    movel([0.119411, -1.390472, -2.566228, -0.755689, 1.570796, 1.690207],accel_mss,speed_ms,0,blend_radius_m)
    movel([0.119247, -1.390171, -2.566445, -0.755774, 1.570796, 1.690044],accel_mss,speed_ms,0,blend_radius_m)
    movel([0.119299, -1.389742, -2.566752, -0.755894, 1.570796, 1.690095],accel_mss,speed_ms,0,blend_radius_m)
    movel([0.119560, -1.389145, -2.567181, -0.756063, 1.570796, 1.690357],accel_mss,speed_ms,0,blend_radius_m)
    movel([0.120675, -1.387270, -2.568525, -0.756595, 1.570796, 1.691472],accel_mss,speed_ms,0,blend_radius_m)
    movel([0.122734, -1.387703, -2.568215, -0.756471, 1.570796, 1.693530],accel_mss,speed_ms,0,blend_radius_m)
    speed_ms = 0.005
    # Splitting Linear movement in 4 (instruction 341: MoveL 309)
    movel([0.122734, -1.385520, -2.567229, -0.759641, 1.570796, 1.693530],accel_mss,speed_ms,0,blend_radius_m)
    movel([0.122734, -1.383346, -2.566239, -0.762804, 1.570796, 1.693530],accel_mss,speed_ms,0,blend_radius_m)
    movel([0.122734, -1.381182, -2.565245, -0.765961, 1.570796, 1.693530],accel_mss,speed_ms,0,blend_radius_m)
    movel([0.122734, -1.379028, -2.564248, -0.769113, 1.570796, 1.693530],accel_mss,speed_ms,0,blend_radius_m)
    speed_ms = 0.040
    # Splitting Linear movement in 18 (instruction 343: MoveL 310)
    movel([0.125073, -1.377791, -2.565121, -0.769477, 1.570796, 1.695869],accel_mss,speed_ms,0,blend_radius_m)
    movel([0.127416, -1.376554, -2.565991, -0.769844, 1.570796, 1.698212],accel_mss,speed_ms,0,blend_radius_m)
    movel([0.129763, -1.375318, -2.566858, -0.770212, 1.570796, 1.700560],accel_mss,speed_ms,0,blend_radius_m)
    movel([0.132116, -1.374083, -2.567723, -0.770583, 1.570796, 1.702912],accel_mss,speed_ms,0,blend_radius_m)
    movel([0.134472, -1.372849, -2.568585, -0.770955, 1.570796, 1.705269],accel_mss,speed_ms,0,blend_radius_m)
    movel([0.136834, -1.371616, -2.569444, -0.771330, 1.570796, 1.707630],accel_mss,speed_ms,0,blend_radius_m)
    movel([0.139200, -1.370383, -2.570300, -0.771706, 1.570796, 1.709996],accel_mss,speed_ms,0,blend_radius_m)
    movel([0.141570, -1.369152, -2.571153, -0.772084, 1.570796, 1.712366],accel_mss,speed_ms,0,blend_radius_m)
    movel([0.143945, -1.367921, -2.572004, -0.772464, 1.570796, 1.714741],accel_mss,speed_ms,0,blend_radius_m)
    movel([0.146324, -1.366692, -2.572852, -0.772845, 1.570796, 1.717121],accel_mss,speed_ms,0,blend_radius_m)
    movel([0.148708, -1.365463, -2.573697, -0.773229, 1.570796, 1.719505],accel_mss,speed_ms,0,blend_radius_m)
    movel([0.151097, -1.364235, -2.574540, -0.773614, 1.570796, 1.721893],accel_mss,speed_ms,0,blend_radius_m)
    movel([0.153490, -1.363008, -2.575379, -0.774001, 1.570796, 1.724286],accel_mss,speed_ms,0,blend_radius_m)
    movel([0.155887, -1.361783, -2.576216, -0.774390, 1.570796, 1.726684],accel_mss,speed_ms,0,blend_radius_m)
    movel([0.158289, -1.360558, -2.577050, -0.774781, 1.570796, 1.729086],accel_mss,speed_ms,0,blend_radius_m)
    movel([0.160696, -1.359335, -2.577881, -0.775173, 1.570796, 1.731492],accel_mss,speed_ms,0,blend_radius_m)
    movel([0.163106, -1.358112, -2.578709, -0.775568, 1.570796, 1.733903],accel_mss,speed_ms,0,blend_radius_m)
    movel([0.165522, -1.356891, -2.579535, -0.775963, 1.570796, 1.736318],accel_mss,speed_ms,0,blend_radius_m)
    speed_ms = 0.005
    # Splitting Linear movement in 6 (instruction 345: MoveL 311)
    movel([0.165522, -1.358351, -2.580216, -0.773822, 1.570796, 1.736318],accel_mss,speed_ms,0,blend_radius_m)
    movel([0.165522, -1.359815, -2.580896, -0.771678, 1.570796, 1.736318],accel_mss,speed_ms,0,blend_radius_m)
    movel([0.165522, -1.361284, -2.581574, -0.769531, 1.570796, 1.736318],accel_mss,speed_ms,0,blend_radius_m)
    movel([0.165522, -1.362758, -2.582250, -0.767381, 1.570796, 1.736318],accel_mss,speed_ms,0,blend_radius_m)
    movel([0.165522, -1.364236, -2.582925, -0.765228, 1.570796, 1.736318],accel_mss,speed_ms,0,blend_radius_m)
    movel([0.165522, -1.365719, -2.583598, -0.763072, 1.570796, 1.736318],accel_mss,speed_ms,0,blend_radius_m)
    speed_ms = 0.035
    movel([0.167244, -1.365978, -2.583421, -0.762990, 1.570796, 1.738040],accel_mss,speed_ms,0,blend_radius_m)
    movel([0.168585, -1.365976, -2.583423, -0.762991, 1.570796, 1.739382],accel_mss,speed_ms,0,blend_radius_m)
    movel([0.169955, -1.365852, -2.583507, -0.763030, 1.570796, 1.740751],accel_mss,speed_ms,0,blend_radius_m)
    movel([0.171344, -1.365613, -2.583670, -0.763105, 1.570796, 1.742141],accel_mss,speed_ms,0,blend_radius_m)
    movel([0.172746, -1.365263, -2.583910, -0.763216, 1.570796, 1.743542],accel_mss,speed_ms,0,blend_radius_m)
    movel([0.174155, -1.364806, -2.584222, -0.763361, 1.570796, 1.744951],accel_mss,speed_ms,0,blend_radius_m)
    movel([0.176950, -1.363591, -2.585050, -0.763747, 1.570796, 1.747746],accel_mss,speed_ms,0,blend_radius_m)
    movel([0.178323, -1.362842, -2.585561, -0.763987, 1.570796, 1.749120],accel_mss,speed_ms,0,blend_radius_m)
    movel([0.180981, -1.361082, -2.586755, -0.764552, 1.570796, 1.751777],accel_mss,speed_ms,0,blend_radius_m)
    movel([0.182252, -1.360079, -2.587434, -0.764876, 1.570796, 1.753048],accel_mss,speed_ms,0,blend_radius_m)
    movel([0.184624, -1.357854, -2.588935, -0.765600, 1.570796, 1.755420],accel_mss,speed_ms,0,blend_radius_m)
    movel([0.185715, -1.356638, -2.589752, -0.765999, 1.570796, 1.756511],accel_mss,speed_ms,0,blend_radius_m)
    movel([0.186729, -1.355358, -2.590610, -0.766421, 1.570796, 1.757525],accel_mss,speed_ms,0,blend_radius_m)
    movel([0.187656, -1.354022, -2.591503, -0.766863, 1.570796, 1.758453],accel_mss,speed_ms,0,blend_radius_m)
    movel([0.188445, -1.352706, -2.592381, -0.767302, 1.570796, 1.759241],accel_mss,speed_ms,0,blend_radius_m)
    movel([0.189111, -1.351390, -2.593256, -0.767743, 1.570796, 1.759907],accel_mss,speed_ms,0,blend_radius_m)
    movel([0.190069, -1.348792, -2.594976, -0.768621, 1.570796, 1.760866],accel_mss,speed_ms,0,blend_radius_m)
    movel([0.190366, -1.347523, -2.595813, -0.769053, 1.570796, 1.761162],accel_mss,speed_ms,0,blend_radius_m)
    movel([0.190585, -1.345090, -2.597412, -0.769888, 1.570796, 1.761381],accel_mss,speed_ms,0,blend_radius_m)
    movel([0.190509, -1.343939, -2.598165, -0.770285, 1.570796, 1.761306],accel_mss,speed_ms,0,blend_radius_m)
    movel([0.189997, -1.341806, -2.599556, -0.771027, 1.570796, 1.760793],accel_mss,speed_ms,0,blend_radius_m)
    movel([0.189557, -1.340837, -2.600186, -0.771366, 1.570796, 1.760353],accel_mss,speed_ms,0,blend_radius_m)
    movel([0.188317, -1.339142, -2.601284, -0.771962, 1.570796, 1.759113],accel_mss,speed_ms,0,blend_radius_m)
    movel([0.187516, -1.338431, -2.601744, -0.772214, 1.570796, 1.758312],accel_mss,speed_ms,0,blend_radius_m)
    movel([0.186599, -1.337819, -2.602140, -0.772431, 1.570796, 1.757395],accel_mss,speed_ms,0,blend_radius_m)
    movel([0.185562, -1.337314, -2.602465, -0.772610, 1.570796, 1.756358],accel_mss,speed_ms,0,blend_radius_m)
    movel([0.183890, -1.336813, -2.602788, -0.772788, 1.570796, 1.754686],accel_mss,speed_ms,0,blend_radius_m)
    movel([0.183257, -1.336822, -2.602782, -0.772785, 1.570796, 1.754053],accel_mss,speed_ms,0,blend_radius_m)
    movel([0.182728, -1.337024, -2.602652, -0.772713, 1.570796, 1.753524],accel_mss,speed_ms,0,blend_radius_m)
    movel([0.182274, -1.337436, -2.602386, -0.772567, 1.570796, 1.753070],accel_mss,speed_ms,0,blend_radius_m)
    movel([0.181874, -1.338070, -2.601977, -0.772342, 1.570796, 1.752671],accel_mss,speed_ms,0,blend_radius_m)
    movel([0.181131, -1.340075, -2.600680, -0.771634, 1.570796, 1.751927],accel_mss,speed_ms,0,blend_radius_m)
    movel([0.182746, -1.340641, -2.600313, -0.771435, 1.570796, 1.753542],accel_mss,speed_ms,0,blend_radius_m)
    movel([0.184246, -1.341473, -2.599772, -0.771144, 1.570796, 1.755043],accel_mss,speed_ms,0,blend_radius_m)
    movel([0.185396, -1.342588, -2.599046, -0.770754, 1.570796, 1.756192],accel_mss,speed_ms,0,blend_radius_m)
    movel([0.186193, -1.343946, -2.598160, -0.770283, 1.570796, 1.756989],accel_mss,speed_ms,0,blend_radius_m)
    movel([0.186629, -1.345508, -2.597137, -0.769744, 1.570796, 1.757425],accel_mss,speed_ms,0,blend_radius_m)
    movel([0.186702, -1.347235, -2.596002, -0.769151, 1.570796, 1.757498],accel_mss,speed_ms,0,blend_radius_m)
    movel([0.186412, -1.349088, -2.594781, -0.768520, 1.570796, 1.757208],accel_mss,speed_ms,0,blend_radius_m)
    movel([0.185753, -1.351031, -2.593494, -0.767864, 1.570796, 1.756550],accel_mss,speed_ms,0,blend_radius_m)
    movel([0.184722, -1.353022, -2.592171, -0.767197, 1.570796, 1.755519],accel_mss,speed_ms,0,blend_radius_m)
    movel([0.183346, -1.354989, -2.590857, -0.766543, 1.570796, 1.754142],accel_mss,speed_ms,0,blend_radius_m)
    movel([0.181729, -1.356786, -2.589652, -0.765950, 1.570796, 1.752525],accel_mss,speed_ms,0,blend_radius_m)
    movel([0.179917, -1.358392, -2.588573, -0.765425, 1.570796, 1.750714],accel_mss,speed_ms,0,blend_radius_m)
    movel([0.177958, -1.359777, -2.587638, -0.764974, 1.570796, 1.748754],accel_mss,speed_ms,0,blend_radius_m)
    movel([0.175895, -1.360914, -2.586869, -0.764606, 1.570796, 1.746691],accel_mss,speed_ms,0,blend_radius_m)
    movel([0.173775, -1.361775, -2.586285, -0.764329, 1.570796, 1.744572],accel_mss,speed_ms,0,blend_radius_m)
    movel([0.171644, -1.362334, -2.585905, -0.764149, 1.570796, 1.742441],accel_mss,speed_ms,0,blend_radius_m)
    movel([0.169547, -1.362562, -2.585751, -0.764076, 1.570796, 1.740343],accel_mss,speed_ms,0,blend_radius_m)
    movel([0.167897, -1.362665, -2.585681, -0.764043, 1.570796, 1.738693],accel_mss,speed_ms,0,blend_radius_m)
    movel([0.167339, -1.362805, -2.585585, -0.763998, 1.570796, 1.738135],accel_mss,speed_ms,0,blend_radius_m)
    movel([0.166903, -1.363048, -2.585420, -0.763921, 1.570796, 1.737699],accel_mss,speed_ms,0,blend_radius_m)
    movel([0.166548, -1.363425, -2.585164, -0.763800, 1.570796, 1.737344],accel_mss,speed_ms,0,blend_radius_m)
    movel([0.166226, -1.363977, -2.584788, -0.763625, 1.570796, 1.737022],accel_mss,speed_ms,0,blend_radius_m)
    movel([0.165522, -1.365719, -2.583598, -0.763072, 1.570796, 1.736318],accel_mss,speed_ms,0,blend_radius_m)
    movel([0.167244, -1.365978, -2.583421, -0.762990, 1.570796, 1.738040],accel_mss,speed_ms,0,blend_radius_m)
    movel([0.167727, -1.365979, -2.583420, -0.762990, 1.570796, 1.738523],accel_mss,speed_ms,0,blend_radius_m)
    speed_ms = 0.005
    # Splitting Linear movement in 4 (instruction 405: MoveL 369)
    movel([0.167727, -1.363756, -2.582411, -0.766222, 1.570796, 1.738523],accel_mss,speed_ms,0,blend_radius_m)
    movel([0.167727, -1.361544, -2.581397, -0.769448, 1.570796, 1.738523],accel_mss,speed_ms,0,blend_radius_m)
    movel([0.167727, -1.359343, -2.580380, -0.772667, 1.570796, 1.738523],accel_mss,speed_ms,0,blend_radius_m)
    movel([0.167727, -1.357152, -2.579359, -0.775879, 1.570796, 1.738523],accel_mss,speed_ms,0,blend_radius_m)
    speed_ms = 0.040
    # Splitting Linear movement in 6 (instruction 407: MoveL 370)
    movel([0.165743, -1.356725, -2.579647, -0.776017, 1.570796, 1.736539],accel_mss,speed_ms,0,blend_radius_m)
    movel([0.163755, -1.356303, -2.579931, -0.776155, 1.570796, 1.734551],accel_mss,speed_ms,0,blend_radius_m)
    movel([0.161764, -1.355886, -2.580213, -0.776291, 1.570796, 1.732560],accel_mss,speed_ms,0,blend_radius_m)
    movel([0.159768, -1.355473, -2.580491, -0.776426, 1.570796, 1.730565],accel_mss,speed_ms,0,blend_radius_m)
    movel([0.157769, -1.355064, -2.580766, -0.776559, 1.570796, 1.728566],accel_mss,speed_ms,0,blend_radius_m)
    movel([0.155767, -1.354660, -2.581037, -0.776692, 1.570796, 1.726563],accel_mss,speed_ms,0,blend_radius_m)
    speed_ms = 0.005
    # Splitting Linear movement in 6 (instruction 409: MoveL 371)
    movel([0.155767, -1.356122, -2.581720, -0.774547, 1.570796, 1.726563],accel_mss,speed_ms,0,blend_radius_m)
    movel([0.155767, -1.357589, -2.582401, -0.772398, 1.570796, 1.726563],accel_mss,speed_ms,0,blend_radius_m)
    movel([0.155767, -1.359061, -2.583081, -0.770247, 1.570796, 1.726563],accel_mss,speed_ms,0,blend_radius_m)
    movel([0.155767, -1.360537, -2.583759, -0.768093, 1.570796, 1.726563],accel_mss,speed_ms,0,blend_radius_m)
    movel([0.155767, -1.362018, -2.584435, -0.765935, 1.570796, 1.726563],accel_mss,speed_ms,0,blend_radius_m)
    movel([0.155767, -1.363504, -2.585110, -0.763775, 1.570796, 1.726563],accel_mss,speed_ms,0,blend_radius_m)
    speed_ms = 0.035
    movel([0.157355, -1.360742, -2.586986, -0.764662, 1.570796, 1.728151],accel_mss,speed_ms,0,blend_radius_m)
    movel([0.158736, -1.358054, -2.588800, -0.765535, 1.570796, 1.729532],accel_mss,speed_ms,0,blend_radius_m)
    movel([0.159906, -1.355440, -2.590555, -0.766394, 1.570796, 1.730702],accel_mss,speed_ms,0,blend_radius_m)
    movel([0.160863, -1.352902, -2.592250, -0.767237, 1.570796, 1.731660],accel_mss,speed_ms,0,blend_radius_m)
    movel([0.161608, -1.350441, -2.593885, -0.768063, 1.570796, 1.732405],accel_mss,speed_ms,0,blend_radius_m)
    movel([0.162137, -1.348053, -2.595464, -0.768872, 1.570796, 1.732933],accel_mss,speed_ms,0,blend_radius_m)
    movel([0.162447, -1.345744, -2.596983, -0.769663, 1.570796, 1.733244],accel_mss,speed_ms,0,blend_radius_m)
    movel([0.162537, -1.343514, -2.598442, -0.770433, 1.570796, 1.733334],accel_mss,speed_ms,0,blend_radius_m)
    movel([0.162403, -1.341361, -2.599845, -0.771183, 1.570796, 1.733200],accel_mss,speed_ms,0,blend_radius_m)
    movel([0.162046, -1.339287, -2.601191, -0.771911, 1.570796, 1.732842],accel_mss,speed_ms,0,blend_radius_m)
    movel([0.161461, -1.337295, -2.602477, -0.772617, 1.570796, 1.732257],accel_mss,speed_ms,0,blend_radius_m)
    movel([0.160647, -1.335385, -2.603706, -0.773298, 1.570796, 1.731443],accel_mss,speed_ms,0,blend_radius_m)
    movel([0.159603, -1.333559, -2.604876, -0.773954, 1.570796, 1.730399],accel_mss,speed_ms,0,blend_radius_m)
    movel([0.158326, -1.331816, -2.605989, -0.774584, 1.570796, 1.729123],accel_mss,speed_ms,0,blend_radius_m)
    movel([0.156817, -1.330161, -2.607041, -0.775187, 1.570796, 1.727613],accel_mss,speed_ms,0,blend_radius_m)
    movel([0.155070, -1.328593, -2.608035, -0.775761, 1.570796, 1.725866],accel_mss,speed_ms,0,blend_radius_m)
    movel([0.156422, -1.327583, -2.608673, -0.776133, 1.570796, 1.727219],accel_mss,speed_ms,0,blend_radius_m)
    movel([0.158344, -1.325960, -2.609696, -0.776733, 1.570796, 1.729140],accel_mss,speed_ms,0,blend_radius_m)
    movel([0.160279, -1.327317, -2.608841, -0.776231, 1.570796, 1.731076],accel_mss,speed_ms,0,blend_radius_m)
    movel([0.161946, -1.328931, -2.607821, -0.775637, 1.570796, 1.732742],accel_mss,speed_ms,0,blend_radius_m)
    movel([0.163339, -1.330774, -2.606652, -0.774963, 1.570796, 1.734136],accel_mss,speed_ms,0,blend_radius_m)
    movel([0.164467, -1.332824, -2.605345, -0.774219, 1.570796, 1.735263],accel_mss,speed_ms,0,blend_radius_m)
    movel([0.165329, -1.335051, -2.603920, -0.773418, 1.570796, 1.736126],accel_mss,speed_ms,0,blend_radius_m)
    movel([0.165930, -1.337434, -2.602388, -0.772567, 1.570796, 1.736726],accel_mss,speed_ms,0,blend_radius_m)
    movel([0.166274, -1.339941, -2.600767, -0.771681, 1.570796, 1.737070],accel_mss,speed_ms,0,blend_radius_m)
    movel([0.166364, -1.342551, -2.599071, -0.770767, 1.570796, 1.737160],accel_mss,speed_ms,0,blend_radius_m)
    movel([0.166202, -1.345238, -2.597314, -0.769836, 1.570796, 1.736998],accel_mss,speed_ms,0,blend_radius_m)
    movel([0.165795, -1.347977, -2.595514, -0.768898, 1.570796, 1.736591],accel_mss,speed_ms,0,blend_radius_m)
    movel([0.165144, -1.350747, -2.593682, -0.767959, 1.570796, 1.735940],accel_mss,speed_ms,0,blend_radius_m)
    movel([0.164254, -1.353520, -2.591838, -0.767031, 1.570796, 1.735050],accel_mss,speed_ms,0,blend_radius_m)
    movel([0.163128, -1.356279, -2.589993, -0.766117, 1.570796, 1.733924],accel_mss,speed_ms,0,blend_radius_m)
    movel([0.161769, -1.358997, -2.588164, -0.765227, 1.570796, 1.732566],accel_mss,speed_ms,0,blend_radius_m)
    movel([0.160179, -1.361655, -2.586367, -0.764368, 1.570796, 1.730976],accel_mss,speed_ms,0,blend_radius_m)
    movel([0.158366, -1.364231, -2.584614, -0.763544, 1.570796, 1.729162],accel_mss,speed_ms,0,blend_radius_m)
    movel([0.155767, -1.363504, -2.585110, -0.763775, 1.570796, 1.726563],accel_mss,speed_ms,0,blend_radius_m)
    movel([0.157104, -1.361176, -2.586691, -0.764522, 1.570796, 1.727901],accel_mss,speed_ms,0,blend_radius_m)
    speed_ms = 0.005
    # Splitting Linear movement in 6 (instruction 448: MoveL 408)
    movel([0.157104, -1.359687, -2.586015, -0.766687, 1.570796, 1.727901],accel_mss,speed_ms,0,blend_radius_m)
    movel([0.157104, -1.358204, -2.585337, -0.768848, 1.570796, 1.727901],accel_mss,speed_ms,0,blend_radius_m)
    movel([0.157104, -1.356725, -2.584657, -0.771007, 1.570796, 1.727901],accel_mss,speed_ms,0,blend_radius_m)
    movel([0.157104, -1.355250, -2.583976, -0.773162, 1.570796, 1.727901],accel_mss,speed_ms,0,blend_radius_m)
    movel([0.157104, -1.353781, -2.583293, -0.775315, 1.570796, 1.727901],accel_mss,speed_ms,0,blend_radius_m)
    movel([0.157104, -1.352316, -2.582608, -0.777465, 1.570796, 1.727901],accel_mss,speed_ms,0,blend_radius_m)
    speed_ms = 0.040
    # Splitting Linear movement in 6 (instruction 450: MoveL 409)
    movel([0.154683, -1.352853, -2.582249, -0.777287, 1.570796, 1.725480],accel_mss,speed_ms,0,blend_radius_m)
    movel([0.152263, -1.353395, -2.581886, -0.777108, 1.570796, 1.723059],accel_mss,speed_ms,0,blend_radius_m)
    movel([0.149843, -1.353940, -2.581520, -0.776928, 1.570796, 1.720639],accel_mss,speed_ms,0,blend_radius_m)
    movel([0.147424, -1.354490, -2.581151, -0.776747, 1.570796, 1.718220],accel_mss,speed_ms,0,blend_radius_m)
    movel([0.145005, -1.355044, -2.580779, -0.776566, 1.570796, 1.715801],accel_mss,speed_ms,0,blend_radius_m)
    movel([0.142587, -1.355603, -2.580403, -0.776383, 1.570796, 1.713383],accel_mss,speed_ms,0,blend_radius_m)
    speed_ms = 0.005
    # Splitting Linear movement in 6 (instruction 452: MoveL 410)
    movel([0.142587, -1.357064, -2.581085, -0.774240, 1.570796, 1.713383],accel_mss,speed_ms,0,blend_radius_m)
    movel([0.142587, -1.358530, -2.581766, -0.772093, 1.570796, 1.713383],accel_mss,speed_ms,0,blend_radius_m)
    movel([0.142587, -1.360001, -2.582445, -0.769944, 1.570796, 1.713383],accel_mss,speed_ms,0,blend_radius_m)
    movel([0.142587, -1.361476, -2.583122, -0.767791, 1.570796, 1.713383],accel_mss,speed_ms,0,blend_radius_m)
    movel([0.142587, -1.362956, -2.583798, -0.765636, 1.570796, 1.713383],accel_mss,speed_ms,0,blend_radius_m)
    movel([0.142587, -1.364440, -2.584472, -0.763477, 1.570796, 1.713383],accel_mss,speed_ms,0,blend_radius_m)
    speed_ms = 0.035
    movel([0.144618, -1.363400, -2.585181, -0.763808, 1.570796, 1.715414],accel_mss,speed_ms,0,blend_radius_m)
    movel([0.145265, -1.363158, -2.585346, -0.763886, 1.570796, 1.716061],accel_mss,speed_ms,0,blend_radius_m)
    movel([0.145714, -1.363112, -2.585377, -0.763900, 1.570796, 1.716510],accel_mss,speed_ms,0,blend_radius_m)
    movel([0.146013, -1.363264, -2.585273, -0.763852, 1.570796, 1.716810],accel_mss,speed_ms,0,blend_radius_m)
    movel([0.146199, -1.363626, -2.585027, -0.763736, 1.570796, 1.716996],accel_mss,speed_ms,0,blend_radius_m)
    movel([0.146391, -1.364992, -2.584095, -0.763302, 1.570796, 1.717188],accel_mss,speed_ms,0,blend_radius_m)
    movel([0.146678, -1.366931, -2.582768, -0.762690, 1.570796, 1.717475],accel_mss,speed_ms,0,blend_radius_m)
    movel([0.147186, -1.368743, -2.581523, -0.762123, 1.570796, 1.717982],accel_mss,speed_ms,0,blend_radius_m)
    movel([0.147904, -1.370420, -2.580367, -0.761602, 1.570796, 1.718700],accel_mss,speed_ms,0,blend_radius_m)
    movel([0.148823, -1.371955, -2.579305, -0.761129, 1.570796, 1.719620],accel_mss,speed_ms,0,blend_radius_m)
    movel([0.149928, -1.373343, -2.578342, -0.760705, 1.570796, 1.720724],accel_mss,speed_ms,0,blend_radius_m)
    movel([0.151213, -1.374577, -2.577483, -0.760329, 1.570796, 1.722009],accel_mss,speed_ms,0,blend_radius_m)
    movel([0.152668, -1.375652, -2.576733, -0.760004, 1.570796, 1.723464],accel_mss,speed_ms,0,blend_radius_m)
    movel([0.154279, -1.376563, -2.576096, -0.759729, 1.570796, 1.725075],accel_mss,speed_ms,0,blend_radius_m)
    movel([0.156039, -1.377302, -2.575579, -0.759508, 1.570796, 1.726835],accel_mss,speed_ms,0,blend_radius_m)
    movel([0.157942, -1.377860, -2.575188, -0.759341, 1.570796, 1.728738],accel_mss,speed_ms,0,blend_radius_m)
    movel([0.159972, -1.378236, -2.574924, -0.759229, 1.570796, 1.730769],accel_mss,speed_ms,0,blend_radius_m)
    movel([0.162127, -1.378415, -2.574799, -0.759176, 1.570796, 1.732924],accel_mss,speed_ms,0,blend_radius_m)
    movel([0.164395, -1.378396, -2.574812, -0.759181, 1.570796, 1.735192],accel_mss,speed_ms,0,blend_radius_m)
    movel([0.166771, -1.378169, -2.574971, -0.759249, 1.570796, 1.737567],accel_mss,speed_ms,0,blend_radius_m)
    movel([0.169243, -1.377725, -2.575282, -0.759381, 1.570796, 1.740039],accel_mss,speed_ms,0,blend_radius_m)
    movel([0.171807, -1.377058, -2.575750, -0.759581, 1.570796, 1.742603],accel_mss,speed_ms,0,blend_radius_m)
    movel([0.174557, -1.376132, -2.576398, -0.759859, 1.570796, 1.745353],accel_mss,speed_ms,0,blend_radius_m)
    movel([0.177244, -1.375031, -2.577167, -0.760192, 1.570796, 1.748040],accel_mss,speed_ms,0,blend_radius_m)
    movel([0.179860, -1.373766, -2.578047, -0.760576, 1.570796, 1.750657],accel_mss,speed_ms,0,blend_radius_m)
    movel([0.182392, -1.372346, -2.579033, -0.761009, 1.570796, 1.753189],accel_mss,speed_ms,0,blend_radius_m)
    movel([0.184834, -1.370780, -2.580118, -0.761491, 1.570796, 1.755630],accel_mss,speed_ms,0,blend_radius_m)
    movel([0.187171, -1.369080, -2.581291, -0.762018, 1.570796, 1.757967],accel_mss,speed_ms,0,blend_radius_m)
    movel([0.189395, -1.367255, -2.582546, -0.762588, 1.570796, 1.760191],accel_mss,speed_ms,0,blend_radius_m)
    movel([0.191497, -1.365311, -2.583877, -0.763201, 1.570796, 1.762293],accel_mss,speed_ms,0,blend_radius_m)
    movel([0.193462, -1.363263, -2.585274, -0.763852, 1.570796, 1.764258],accel_mss,speed_ms,0,blend_radius_m)
    movel([0.195284, -1.361118, -2.586730, -0.764540, 1.570796, 1.766080],accel_mss,speed_ms,0,blend_radius_m)
    movel([0.196947, -1.358890, -2.588237, -0.765262, 1.570796, 1.767743],accel_mss,speed_ms,0,blend_radius_m)
    movel([0.198441, -1.356584, -2.589788, -0.766017, 1.570796, 1.769238],accel_mss,speed_ms,0,blend_radius_m)
    movel([0.199751, -1.354218, -2.591373, -0.766799, 1.570796, 1.770547],accel_mss,speed_ms,0,blend_radius_m)
    movel([0.200870, -1.351797, -2.592986, -0.767607, 1.570796, 1.771666],accel_mss,speed_ms,0,blend_radius_m)
    movel([0.201780, -1.349333, -2.594619, -0.768437, 1.570796, 1.772576],accel_mss,speed_ms,0,blend_radius_m)
    movel([0.202469, -1.346842, -2.596261, -0.769286, 1.570796, 1.773266],accel_mss,speed_ms,0,blend_radius_m)
    movel([0.202849, -1.344806, -2.597598, -0.769986, 1.570796, 1.773645],accel_mss,speed_ms,0,blend_radius_m)
    movel([0.203044, -1.342836, -2.598885, -0.770668, 1.570796, 1.773841],accel_mss,speed_ms,0,blend_radius_m)
    movel([0.203058, -1.340938, -2.600120, -0.771331, 1.570796, 1.773854],accel_mss,speed_ms,0,blend_radius_m)
    movel([0.202894, -1.339124, -2.601296, -0.771969, 1.570796, 1.773690],accel_mss,speed_ms,0,blend_radius_m)
    movel([0.202553, -1.337396, -2.602412, -0.772581, 1.570796, 1.773349],accel_mss,speed_ms,0,blend_radius_m)
    movel([0.202041, -1.335767, -2.603461, -0.773161, 1.570796, 1.772837],accel_mss,speed_ms,0,blend_radius_m)
    movel([0.201360, -1.334242, -2.604439, -0.773708, 1.570796, 1.772156],accel_mss,speed_ms,0,blend_radius_m)
    movel([0.200513, -1.332830, -2.605342, -0.774217, 1.570796, 1.771309],accel_mss,speed_ms,0,blend_radius_m)
    movel([0.199505, -1.331537, -2.606166, -0.774686, 1.570796, 1.770301],accel_mss,speed_ms,0,blend_radius_m)
    movel([0.198339, -1.330373, -2.606906, -0.775110, 1.570796, 1.769136],accel_mss,speed_ms,0,blend_radius_m)
    movel([0.197021, -1.329344, -2.607559, -0.775486, 1.570796, 1.767817],accel_mss,speed_ms,0,blend_radius_m)
    movel([0.195555, -1.328459, -2.608119, -0.775810, 1.570796, 1.766352],accel_mss,speed_ms,0,blend_radius_m)
    movel([0.193946, -1.327726, -2.608583, -0.776080, 1.570796, 1.764742],accel_mss,speed_ms,0,blend_radius_m)
    movel([0.192197, -1.327150, -2.608947, -0.776293, 1.570796, 1.762993],accel_mss,speed_ms,0,blend_radius_m)
    movel([0.190314, -1.326740, -2.609205, -0.776444, 1.570796, 1.761110],accel_mss,speed_ms,0,blend_radius_m)
    movel([0.188302, -1.326505, -2.609353, -0.776531, 1.570796, 1.759098],accel_mss,speed_ms,0,blend_radius_m)
    movel([0.186033, -1.326287, -2.609490, -0.776612, 1.570796, 1.756829],accel_mss,speed_ms,0,blend_radius_m)
    movel([0.186699, -1.324329, -2.610721, -0.777339, 1.570796, 1.757495],accel_mss,speed_ms,0,blend_radius_m)
    movel([0.187062, -1.323682, -2.611126, -0.777581, 1.570796, 1.757858],accel_mss,speed_ms,0,blend_radius_m)
    movel([0.187486, -1.323227, -2.611411, -0.777751, 1.570796, 1.758283],accel_mss,speed_ms,0,blend_radius_m)
    movel([0.188004, -1.322935, -2.611594, -0.777861, 1.570796, 1.758800],accel_mss,speed_ms,0,blend_radius_m)
    movel([0.188643, -1.322782, -2.611689, -0.777918, 1.570796, 1.759439],accel_mss,speed_ms,0,blend_radius_m)
    movel([0.190414, -1.322802, -2.611676, -0.777910, 1.570796, 1.761210],accel_mss,speed_ms,0,blend_radius_m)
    movel([0.192754, -1.323116, -2.611480, -0.777793, 1.570796, 1.763550],accel_mss,speed_ms,0,blend_radius_m)
    movel([0.194935, -1.323635, -2.611155, -0.777598, 1.570796, 1.765732],accel_mss,speed_ms,0,blend_radius_m)
    movel([0.196955, -1.324350, -2.610707, -0.777331, 1.570796, 1.767752],accel_mss,speed_ms,0,blend_radius_m)
    movel([0.198804, -1.325254, -2.610140, -0.776995, 1.570796, 1.769600],accel_mss,speed_ms,0,blend_radius_m)
    movel([0.200476, -1.326336, -2.609459, -0.776593, 1.570796, 1.771272],accel_mss,speed_ms,0,blend_radius_m)
    movel([0.201971, -1.327585, -2.608672, -0.776132, 1.570796, 1.772767],accel_mss,speed_ms,0,blend_radius_m)
    movel([0.203277, -1.328995, -2.607780, -0.775614, 1.570796, 1.774073],accel_mss,speed_ms,0,blend_radius_m)
    movel([0.204395, -1.330550, -2.606794, -0.775045, 1.570796, 1.775192],accel_mss,speed_ms,0,blend_radius_m)
    movel([0.205318, -1.332246, -2.605714, -0.774428, 1.570796, 1.776115],accel_mss,speed_ms,0,blend_radius_m)
    movel([0.206044, -1.334068, -2.604550, -0.773771, 1.570796, 1.776841],accel_mss,speed_ms,0,blend_radius_m)
    movel([0.206568, -1.336009, -2.603305, -0.773075, 1.570796, 1.777365],accel_mss,speed_ms,0,blend_radius_m)
    movel([0.206883, -1.338059, -2.601984, -0.772345, 1.570796, 1.777680],accel_mss,speed_ms,0,blend_radius_m)
    movel([0.206991, -1.340206, -2.600596, -0.771588, 1.570796, 1.777788],accel_mss,speed_ms,0,blend_radius_m)
    movel([0.206884, -1.342444, -2.599140, -0.770805, 1.570796, 1.777681],accel_mss,speed_ms,0,blend_radius_m)
    movel([0.206563, -1.344758, -2.597629, -0.770002, 1.570796, 1.777359],accel_mss,speed_ms,0,blend_radius_m)
    movel([0.206022, -1.347143, -2.596063, -0.769183, 1.570796, 1.776818],accel_mss,speed_ms,0,blend_radius_m)
    movel([0.205270, -1.349550, -2.594475, -0.768364, 1.570796, 1.776066],accel_mss,speed_ms,0,blend_radius_m)
    movel([0.204329, -1.351941, -2.592890, -0.767558, 1.570796, 1.775125],accel_mss,speed_ms,0,blend_radius_m)
    movel([0.203206, -1.354307, -2.591313, -0.766769, 1.570796, 1.774003],accel_mss,speed_ms,0,blend_radius_m)
    movel([0.201915, -1.356634, -2.589755, -0.766000, 1.570796, 1.772711],accel_mss,speed_ms,0,blend_radius_m)
    movel([0.200464, -1.358916, -2.588219, -0.765254, 1.570796, 1.771260],accel_mss,speed_ms,0,blend_radius_m)
    movel([0.198867, -1.361141, -2.586715, -0.764533, 1.570796, 1.769664],accel_mss,speed_ms,0,blend_radius_m)
    movel([0.197131, -1.363302, -2.585247, -0.763839, 1.570796, 1.767927],accel_mss,speed_ms,0,blend_radius_m)
    movel([0.195269, -1.365387, -2.583825, -0.763177, 1.570796, 1.766065],accel_mss,speed_ms,0,blend_radius_m)
    movel([0.193289, -1.367390, -2.582453, -0.762546, 1.570796, 1.764085],accel_mss,speed_ms,0,blend_radius_m)
    movel([0.191199, -1.369302, -2.581138, -0.761949, 1.570796, 1.761995],accel_mss,speed_ms,0,blend_radius_m)
    movel([0.189008, -1.371111, -2.579889, -0.761389, 1.570796, 1.759805],accel_mss,speed_ms,0,blend_radius_m)
    movel([0.186730, -1.372813, -2.578709, -0.760866, 1.570796, 1.757527],accel_mss,speed_ms,0,blend_radius_m)
    movel([0.184369, -1.374394, -2.577610, -0.760385, 1.570796, 1.755166],accel_mss,speed_ms,0,blend_radius_m)
    movel([0.181935, -1.375853, -2.576593, -0.759943, 1.570796, 1.752731],accel_mss,speed_ms,0,blend_radius_m)
    movel([0.179436, -1.377174, -2.575669, -0.759546, 1.570796, 1.750233],accel_mss,speed_ms,0,blend_radius_m)
    movel([0.176882, -1.378351, -2.574844, -0.759195, 1.570796, 1.747678],accel_mss,speed_ms,0,blend_radius_m)
    movel([0.174330, -1.379357, -2.574136, -0.758895, 1.570796, 1.745127],accel_mss,speed_ms,0,blend_radius_m)
    movel([0.171808, -1.380183, -2.573555, -0.758651, 1.570796, 1.742604],accel_mss,speed_ms,0,blend_radius_m)
    movel([0.169325, -1.380833, -2.573097, -0.758460, 1.570796, 1.740121],accel_mss,speed_ms,0,blend_radius_m)
    movel([0.166894, -1.381304, -2.572764, -0.758321, 1.570796, 1.737691],accel_mss,speed_ms,0,blend_radius_m)
    movel([0.164518, -1.381602, -2.572553, -0.758233, 1.570796, 1.735315],accel_mss,speed_ms,0,blend_radius_m)
    movel([0.162212, -1.381729, -2.572463, -0.758196, 1.570796, 1.733009],accel_mss,speed_ms,0,blend_radius_m)
    movel([0.159981, -1.381688, -2.572493, -0.758208, 1.570796, 1.730778],accel_mss,speed_ms,0,blend_radius_m)
    movel([0.157837, -1.381474, -2.572644, -0.758271, 1.570796, 1.728633],accel_mss,speed_ms,0,blend_radius_m)
    movel([0.155786, -1.381095, -2.572911, -0.758382, 1.570796, 1.726582],accel_mss,speed_ms,0,blend_radius_m)
    movel([0.153843, -1.380549, -2.573297, -0.758543, 1.570796, 1.724639],accel_mss,speed_ms,0,blend_radius_m)
    movel([0.152016, -1.379836, -2.573800, -0.758754, 1.570796, 1.722813],accel_mss,speed_ms,0,blend_radius_m)
    movel([0.150314, -1.378957, -2.574418, -0.759014, 1.570796, 1.721111],accel_mss,speed_ms,0,blend_radius_m)
    movel([0.148748, -1.377914, -2.575150, -0.759325, 1.570796, 1.719545],accel_mss,speed_ms,0,blend_radius_m)
    movel([0.147329, -1.376704, -2.575998, -0.759687, 1.570796, 1.718125],accel_mss,speed_ms,0,blend_radius_m)
    movel([0.146068, -1.375329, -2.576959, -0.760101, 1.570796, 1.716865],accel_mss,speed_ms,0,blend_radius_m)
    movel([0.144973, -1.373788, -2.578032, -0.760569, 1.570796, 1.715770],accel_mss,speed_ms,0,blend_radius_m)
    movel([0.143879, -1.371725, -2.579464, -0.761200, 1.570796, 1.714675],accel_mss,speed_ms,0,blend_radius_m)
    movel([0.143082, -1.369495, -2.581005, -0.761889, 1.570796, 1.713878],accel_mss,speed_ms,0,blend_radius_m)
    movel([0.142634, -1.367074, -2.582670, -0.762645, 1.570796, 1.713430],accel_mss,speed_ms,0,blend_radius_m)
    movel([0.142587, -1.364440, -2.584472, -0.763477, 1.570796, 1.713383],accel_mss,speed_ms,0,blend_radius_m)
    movel([0.144618, -1.363400, -2.585181, -0.763808, 1.570796, 1.715414],accel_mss,speed_ms,0,blend_radius_m)
    movel([0.145130, -1.363209, -2.585311, -0.763869, 1.570796, 1.715926],accel_mss,speed_ms,0,blend_radius_m)
    speed_ms = 0.005
    # Splitting Linear movement in 4 (instruction 570: MoveL 526)
    movel([0.145130, -1.360982, -2.584298, -0.767110, 1.570796, 1.715926],accel_mss,speed_ms,0,blend_radius_m)
    movel([0.145130, -1.358765, -2.583281, -0.770343, 1.570796, 1.715926],accel_mss,speed_ms,0,blend_radius_m)
    movel([0.145130, -1.356559, -2.582261, -0.773569, 1.570796, 1.715926],accel_mss,speed_ms,0,blend_radius_m)
    movel([0.145130, -1.354363, -2.581237, -0.776789, 1.570796, 1.715926],accel_mss,speed_ms,0,blend_radius_m)
    speed_ms = 0.040
    # Splitting Linear movement in 10 (instruction 572: MoveL 527)
    movel([0.142834, -1.354927, -2.580858, -0.776604, 1.570796, 1.713630],accel_mss,speed_ms,0,blend_radius_m)
    movel([0.140539, -1.355494, -2.580476, -0.776419, 1.570796, 1.711335],accel_mss,speed_ms,0,blend_radius_m)
    movel([0.138244, -1.356065, -2.580092, -0.776232, 1.570796, 1.709040],accel_mss,speed_ms,0,blend_radius_m)
    movel([0.135951, -1.356640, -2.579704, -0.776045, 1.570796, 1.706747],accel_mss,speed_ms,0,blend_radius_m)
    movel([0.133658, -1.357218, -2.579314, -0.775857, 1.570796, 1.704454],accel_mss,speed_ms,0,blend_radius_m)
    movel([0.131366, -1.357800, -2.578921, -0.775669, 1.570796, 1.702162],accel_mss,speed_ms,0,blend_radius_m)
    movel([0.129075, -1.358385, -2.578525, -0.775479, 1.570796, 1.699871],accel_mss,speed_ms,0,blend_radius_m)
    movel([0.126784, -1.358974, -2.578126, -0.775289, 1.570796, 1.697581],accel_mss,speed_ms,0,blend_radius_m)
    movel([0.124495, -1.359567, -2.577724, -0.775099, 1.570796, 1.695291],accel_mss,speed_ms,0,blend_radius_m)
    movel([0.122207, -1.360163, -2.577319, -0.774908, 1.570796, 1.693003],accel_mss,speed_ms,0,blend_radius_m)
    speed_ms = 0.005
    # Splitting Linear movement in 4 (instruction 574: MoveL 528)
    movel([0.122207, -1.362349, -2.578336, -0.771704, 1.570796, 1.693003],accel_mss,speed_ms,0,blend_radius_m)
    movel([0.122207, -1.364545, -2.579350, -0.768493, 1.570796, 1.693003],accel_mss,speed_ms,0,blend_radius_m)
    movel([0.122207, -1.366752, -2.580361, -0.765276, 1.570796, 1.693003],accel_mss,speed_ms,0,blend_radius_m)
    movel([0.122207, -1.368969, -2.581367, -0.762053, 1.570796, 1.693003],accel_mss,speed_ms,0,blend_radius_m)
    speed_ms = 0.035
    movel([0.120628, -1.371920, -2.579329, -0.761140, 1.570796, 1.691424],accel_mss,speed_ms,0,blend_radius_m)
    movel([0.119214, -1.371762, -2.579438, -0.761188, 1.570796, 1.690010],accel_mss,speed_ms,0,blend_radius_m)
    movel([0.117940, -1.371473, -2.579638, -0.761277, 1.570796, 1.688737],accel_mss,speed_ms,0,blend_radius_m)
    movel([0.116802, -1.371057, -2.579926, -0.761406, 1.570796, 1.687599],accel_mss,speed_ms,0,blend_radius_m)
    movel([0.115794, -1.370517, -2.580299, -0.761572, 1.570796, 1.686590],accel_mss,speed_ms,0,blend_radius_m)
    movel([0.114907, -1.369857, -2.580755, -0.761777, 1.570796, 1.685704],accel_mss,speed_ms,0,blend_radius_m)
    movel([0.114139, -1.369082, -2.581290, -0.762018, 1.570796, 1.684935],accel_mss,speed_ms,0,blend_radius_m)
    movel([0.113482, -1.368197, -2.581899, -0.762294, 1.570796, 1.684278],accel_mss,speed_ms,0,blend_radius_m)
    movel([0.112927, -1.367203, -2.582581, -0.762605, 1.570796, 1.683724],accel_mss,speed_ms,0,blend_radius_m)
    movel([0.112291, -1.365333, -2.583862, -0.763194, 1.570796, 1.683087],accel_mss,speed_ms,0,blend_radius_m)
    movel([0.112068, -1.363283, -2.585260, -0.763846, 1.570796, 1.682864],accel_mss,speed_ms,0,blend_radius_m)
    movel([0.112247, -1.361095, -2.586746, -0.764548, 1.570796, 1.683043],accel_mss,speed_ms,0,blend_radius_m)
    movel([0.112813, -1.358816, -2.588287, -0.765286, 1.570796, 1.683610],accel_mss,speed_ms,0,blend_radius_m)
    movel([0.113756, -1.356481, -2.589857, -0.766050, 1.570796, 1.684553],accel_mss,speed_ms,0,blend_radius_m)
    movel([0.115059, -1.354143, -2.591423, -0.766823, 1.570796, 1.685855],accel_mss,speed_ms,0,blend_radius_m)
    movel([0.116712, -1.351839, -2.592957, -0.767592, 1.570796, 1.687508],accel_mss,speed_ms,0,blend_radius_m)
    movel([0.118694, -1.349622, -2.594428, -0.768340, 1.570796, 1.689491],accel_mss,speed_ms,0,blend_radius_m)
    movel([0.120927, -1.347589, -2.595769, -0.769030, 1.570796, 1.691723],accel_mss,speed_ms,0,blend_radius_m)
    movel([0.123311, -1.345817, -2.596935, -0.769637, 1.570796, 1.694107],accel_mss,speed_ms,0,blend_radius_m)
    movel([0.125806, -1.344321, -2.597915, -0.770153, 1.570796, 1.696602],accel_mss,speed_ms,0,blend_radius_m)
    movel([0.128360, -1.343128, -2.598694, -0.770567, 1.570796, 1.699157],accel_mss,speed_ms,0,blend_radius_m)
    movel([0.130924, -1.342257, -2.599262, -0.770870, 1.570796, 1.701720],accel_mss,speed_ms,0,blend_radius_m)
    movel([0.133454, -1.341729, -2.599606, -0.771054, 1.570796, 1.704250],accel_mss,speed_ms,0,blend_radius_m)
    movel([0.135896, -1.341564, -2.599713, -0.771112, 1.570796, 1.706692],accel_mss,speed_ms,0,blend_radius_m)
    movel([0.138205, -1.341781, -2.599572, -0.771036, 1.570796, 1.709002],accel_mss,speed_ms,0,blend_radius_m)
    movel([0.140282, -1.342388, -2.599177, -0.770824, 1.570796, 1.711078],accel_mss,speed_ms,0,blend_radius_m)
    movel([0.142032, -1.343350, -2.598549, -0.770489, 1.570796, 1.712829],accel_mss,speed_ms,0,blend_radius_m)
    movel([0.143439, -1.344635, -2.597709, -0.770045, 1.570796, 1.714235],accel_mss,speed_ms,0,blend_radius_m)
    movel([0.144488, -1.346208, -2.596678, -0.769503, 1.570796, 1.715284],accel_mss,speed_ms,0,blend_radius_m)
    movel([0.145165, -1.348036, -2.595475, -0.768878, 1.570796, 1.715961],accel_mss,speed_ms,0,blend_radius_m)
    movel([0.145455, -1.350083, -2.594123, -0.768184, 1.570796, 1.716251],accel_mss,speed_ms,0,blend_radius_m)
    movel([0.145344, -1.352316, -2.592640, -0.767432, 1.570796, 1.716141],accel_mss,speed_ms,0,blend_radius_m)
    movel([0.144824, -1.354700, -2.591050, -0.766639, 1.570796, 1.715620],accel_mss,speed_ms,0,blend_radius_m)
    movel([0.144168, -1.356513, -2.589836, -0.766040, 1.570796, 1.714964],accel_mss,speed_ms,0,blend_radius_m)
    movel([0.143799, -1.357128, -2.589423, -0.765838, 1.570796, 1.714595],accel_mss,speed_ms,0,blend_radius_m)
    movel([0.143353, -1.357588, -2.589114, -0.765687, 1.570796, 1.714149],accel_mss,speed_ms,0,blend_radius_m)
    movel([0.142793, -1.357923, -2.588888, -0.765578, 1.570796, 1.713589],accel_mss,speed_ms,0,blend_radius_m)
    movel([0.142084, -1.358161, -2.588728, -0.765500, 1.570796, 1.712880],accel_mss,speed_ms,0,blend_radius_m)
    movel([0.140076, -1.358461, -2.588526, -0.765402, 1.570796, 1.710872],accel_mss,speed_ms,0,blend_radius_m)
    movel([0.140788, -1.355200, -2.590716, -0.766473, 1.570796, 1.711585],accel_mss,speed_ms,0,blend_radius_m)
    movel([0.141097, -1.352421, -2.592571, -0.767398, 1.570796, 1.711893],accel_mss,speed_ms,0,blend_radius_m)
    movel([0.140994, -1.350112, -2.594103, -0.768174, 1.570796, 1.711790],accel_mss,speed_ms,0,blend_radius_m)
    movel([0.140462, -1.348263, -2.595325, -0.768801, 1.570796, 1.711258],accel_mss,speed_ms,0,blend_radius_m)
    movel([0.140033, -1.347506, -2.595824, -0.769059, 1.570796, 1.710829],accel_mss,speed_ms,0,blend_radius_m)
    movel([0.139494, -1.346858, -2.596251, -0.769280, 1.570796, 1.710290],accel_mss,speed_ms,0,blend_radius_m)
    movel([0.138842, -1.346318, -2.596606, -0.769465, 1.570796, 1.709638],accel_mss,speed_ms,0,blend_radius_m)
    movel([0.137202, -1.345554, -2.597107, -0.769728, 1.570796, 1.707998],accel_mss,speed_ms,0,blend_radius_m)
    movel([0.136209, -1.345326, -2.597257, -0.769806, 1.570796, 1.707005],accel_mss,speed_ms,0,blend_radius_m)
    movel([0.133874, -1.345167, -2.597361, -0.769861, 1.570796, 1.704670],accel_mss,speed_ms,0,blend_radius_m)
    movel([0.131737, -1.345382, -2.597220, -0.769787, 1.570796, 1.702534],accel_mss,speed_ms,0,blend_radius_m)
    movel([0.129547, -1.345948, -2.596849, -0.769593, 1.570796, 1.700343],accel_mss,speed_ms,0,blend_radius_m)
    movel([0.127354, -1.346830, -2.596269, -0.769290, 1.570796, 1.698150],accel_mss,speed_ms,0,blend_radius_m)
    movel([0.125210, -1.347998, -2.595500, -0.768891, 1.570796, 1.696007],accel_mss,speed_ms,0,blend_radius_m)
    movel([0.123173, -1.349416, -2.594564, -0.768409, 1.570796, 1.693969],accel_mss,speed_ms,0,blend_radius_m)
    movel([0.121287, -1.351053, -2.593479, -0.767856, 1.570796, 1.692083],accel_mss,speed_ms,0,blend_radius_m)
    movel([0.119605, -1.352873, -2.592270, -0.767246, 1.570796, 1.690401],accel_mss,speed_ms,0,blend_radius_m)
    movel([0.118176, -1.354846, -2.590953, -0.766590, 1.570796, 1.688972],accel_mss,speed_ms,0,blend_radius_m)
    movel([0.116876, -1.357206, -2.589370, -0.765812, 1.570796, 1.687673],accel_mss,speed_ms,0,blend_radius_m)
    movel([0.116086, -1.359360, -2.587920, -0.765109, 1.570796, 1.686883],accel_mss,speed_ms,0,blend_radius_m)
    movel([0.115884, -1.360363, -2.587241, -0.764784, 1.570796, 1.686680],accel_mss,speed_ms,0,blend_radius_m)
    movel([0.115866, -1.362242, -2.585968, -0.764179, 1.570796, 1.686662],accel_mss,speed_ms,0,blend_radius_m)
    movel([0.116049, -1.363120, -2.585371, -0.763898, 1.570796, 1.686846],accel_mss,speed_ms,0,blend_radius_m)
    movel([0.116806, -1.364762, -2.584252, -0.763375, 1.570796, 1.687602],accel_mss,speed_ms,0,blend_radius_m)
    movel([0.118084, -1.366274, -2.583218, -0.762897, 1.570796, 1.688880],accel_mss,speed_ms,0,blend_radius_m)
    movel([0.119883, -1.367669, -2.582262, -0.762459, 1.570796, 1.690680],accel_mss,speed_ms,0,blend_radius_m)
    movel([0.122207, -1.368969, -2.581367, -0.762053, 1.570796, 1.693003],accel_mss,speed_ms,0,blend_radius_m)
    movel([0.120970, -1.371277, -2.579774, -0.761338, 1.570796, 1.691767],accel_mss,speed_ms,0,blend_radius_m)
    speed_ms = 0.005
    # Splitting Linear movement in 6 (instruction 644: MoveL 596)
    movel([0.120970, -1.369801, -2.579105, -0.763483, 1.570796, 1.691767],accel_mss,speed_ms,0,blend_radius_m)
    movel([0.120970, -1.368329, -2.578435, -0.765626, 1.570796, 1.691767],accel_mss,speed_ms,0,blend_radius_m)
    movel([0.120970, -1.366861, -2.577762, -0.767765, 1.570796, 1.691767],accel_mss,speed_ms,0,blend_radius_m)
    movel([0.120970, -1.365398, -2.577088, -0.769902, 1.570796, 1.691767],accel_mss,speed_ms,0,blend_radius_m)
    movel([0.120970, -1.363940, -2.576413, -0.772036, 1.570796, 1.691767],accel_mss,speed_ms,0,blend_radius_m)
    movel([0.120970, -1.362487, -2.575736, -0.774167, 1.570796, 1.691767],accel_mss,speed_ms,0,blend_radius_m)
    speed_ms = 0.040
    # Splitting Linear movement in 18 (instruction 646: MoveL 597)
    movel([0.120281, -1.360880, -2.576831, -0.774678, 1.570796, 1.691078],accel_mss,speed_ms,0,blend_radius_m)
    movel([0.119589, -1.359271, -2.577924, -0.775194, 1.570796, 1.690386],accel_mss,speed_ms,0,blend_radius_m)
    movel([0.118894, -1.357660, -2.579015, -0.775714, 1.570796, 1.689691],accel_mss,speed_ms,0,blend_radius_m)
    movel([0.118196, -1.356047, -2.580104, -0.776238, 1.570796, 1.688993],accel_mss,speed_ms,0,blend_radius_m)
    movel([0.117496, -1.354432, -2.581190, -0.776767, 1.570796, 1.688292],accel_mss,speed_ms,0,blend_radius_m)
    movel([0.116792, -1.352815, -2.582275, -0.777299, 1.570796, 1.687588],accel_mss,speed_ms,0,blend_radius_m)
    movel([0.116085, -1.351195, -2.583357, -0.777837, 1.570796, 1.686882],accel_mss,speed_ms,0,blend_radius_m)
    movel([0.115376, -1.349574, -2.584437, -0.778378, 1.570796, 1.686172],accel_mss,speed_ms,0,blend_radius_m)
    movel([0.114663, -1.347950, -2.585515, -0.778924, 1.570796, 1.685460],accel_mss,speed_ms,0,blend_radius_m)
    movel([0.113948, -1.346324, -2.586591, -0.779475, 1.570796, 1.684744],accel_mss,speed_ms,0,blend_radius_m)
    movel([0.113229, -1.344696, -2.587664, -0.780029, 1.570796, 1.684025],accel_mss,speed_ms,0,blend_radius_m)
    movel([0.112508, -1.343065, -2.588736, -0.780588, 1.570796, 1.683304],accel_mss,speed_ms,0,blend_radius_m)
    movel([0.111783, -1.341433, -2.589805, -0.781152, 1.570796, 1.682579],accel_mss,speed_ms,0,blend_radius_m)
    movel([0.111055, -1.339798, -2.590871, -0.781719, 1.570796, 1.681852],accel_mss,speed_ms,0,blend_radius_m)
    movel([0.110324, -1.338161, -2.591936, -0.782292, 1.570796, 1.681121],accel_mss,speed_ms,0,blend_radius_m)
    movel([0.109590, -1.336522, -2.592998, -0.782868, 1.570796, 1.680387],accel_mss,speed_ms,0,blend_radius_m)
    movel([0.108853, -1.334881, -2.594059, -0.783449, 1.570796, 1.679650],accel_mss,speed_ms,0,blend_radius_m)
    movel([0.108113, -1.333238, -2.595116, -0.784034, 1.570796, 1.678910],accel_mss,speed_ms,0,blend_radius_m)
    speed_ms = 0.005
    # Splitting Linear movement in 6 (instruction 648: MoveL 598)
    movel([0.108113, -1.334723, -2.595815, -0.781850, 1.570796, 1.678910],accel_mss,speed_ms,0,blend_radius_m)
    movel([0.108113, -1.336214, -2.596512, -0.779663, 1.570796, 1.678910],accel_mss,speed_ms,0,blend_radius_m)
    movel([0.108113, -1.337709, -2.597208, -0.777473, 1.570796, 1.678910],accel_mss,speed_ms,0,blend_radius_m)
    movel([0.108113, -1.339209, -2.597901, -0.775279, 1.570796, 1.678910],accel_mss,speed_ms,0,blend_radius_m)
    movel([0.108113, -1.340714, -2.598593, -0.773082, 1.570796, 1.678910],accel_mss,speed_ms,0,blend_radius_m)
    movel([0.108113, -1.342224, -2.599284, -0.770881, 1.570796, 1.678910],accel_mss,speed_ms,0,blend_radius_m)
    speed_ms = 0.035
    movel([0.106316, -1.344176, -2.598009, -0.770203, 1.570796, 1.677112],accel_mss,speed_ms,0,blend_radius_m)
    movel([0.104661, -1.346139, -2.596723, -0.769527, 1.570796, 1.675458],accel_mss,speed_ms,0,blend_radius_m)
    movel([0.103151, -1.348105, -2.595429, -0.768854, 1.570796, 1.673947],accel_mss,speed_ms,0,blend_radius_m)
    movel([0.101779, -1.350073, -2.594129, -0.768187, 1.570796, 1.672575],accel_mss,speed_ms,0,blend_radius_m)
    movel([0.100547, -1.352034, -2.592828, -0.767527, 1.570796, 1.671344],accel_mss,speed_ms,0,blend_radius_m)
    movel([0.099454, -1.353987, -2.591527, -0.766875, 1.570796, 1.670250],accel_mss,speed_ms,0,blend_radius_m)
    movel([0.098494, -1.355925, -2.590231, -0.766234, 1.570796, 1.669290],accel_mss,speed_ms,0,blend_radius_m)
    movel([0.097668, -1.357843, -2.588942, -0.765604, 1.570796, 1.668464],accel_mss,speed_ms,0,blend_radius_m)
    movel([0.096975, -1.359738, -2.587665, -0.764987, 1.570796, 1.667771],accel_mss,speed_ms,0,blend_radius_m)
    movel([0.096414, -1.361603, -2.586402, -0.764384, 1.570796, 1.667210],accel_mss,speed_ms,0,blend_radius_m)
    movel([0.095669, -1.365229, -2.583933, -0.763227, 1.570796, 1.666466],accel_mss,speed_ms,0,blend_radius_m)
    movel([0.095485, -1.366984, -2.582732, -0.762673, 1.570796, 1.666281],accel_mss,speed_ms,0,blend_radius_m)
    movel([0.095485, -1.370347, -2.580417, -0.761625, 1.570796, 1.666281],accel_mss,speed_ms,0,blend_radius_m)
    movel([0.095663, -1.371951, -2.579308, -0.761131, 1.570796, 1.666459],accel_mss,speed_ms,0,blend_radius_m)
    movel([0.096371, -1.374980, -2.577202, -0.760207, 1.570796, 1.667167],accel_mss,speed_ms,0,blend_radius_m)
    movel([0.096895, -1.376399, -2.576211, -0.759779, 1.570796, 1.667692],accel_mss,speed_ms,0,blend_radius_m)
    movel([0.098286, -1.379018, -2.574375, -0.758996, 1.570796, 1.669082],accel_mss,speed_ms,0,blend_radius_m)
    movel([0.099145, -1.380214, -2.573533, -0.758642, 1.570796, 1.669941],accel_mss,speed_ms,0,blend_radius_m)
    movel([0.101187, -1.382355, -2.572020, -0.758013, 1.570796, 1.671984],accel_mss,speed_ms,0,blend_radius_m)
    movel([0.102370, -1.383294, -2.571355, -0.757739, 1.570796, 1.673166],accel_mss,speed_ms,0,blend_radius_m)
    movel([0.103656, -1.384139, -2.570755, -0.757494, 1.570796, 1.674453],accel_mss,speed_ms,0,blend_radius_m)
    movel([0.105046, -1.384888, -2.570223, -0.757278, 1.570796, 1.675842],accel_mss,speed_ms,0,blend_radius_m)
    movel([0.106539, -1.385533, -2.569764, -0.757092, 1.570796, 1.677335],accel_mss,speed_ms,0,blend_radius_m)
    movel([0.108133, -1.386075, -2.569377, -0.756936, 1.570796, 1.678929],accel_mss,speed_ms,0,blend_radius_m)
    movel([0.109829, -1.386506, -2.569070, -0.756813, 1.570796, 1.680626],accel_mss,speed_ms,0,blend_radius_m)
    movel([0.111627, -1.386823, -2.568843, -0.756722, 1.570796, 1.682423],accel_mss,speed_ms,0,blend_radius_m)
    movel([0.113523, -1.387023, -2.568701, -0.756665, 1.570796, 1.684320],accel_mss,speed_ms,0,blend_radius_m)
    movel([0.112735, -1.388822, -2.567413, -0.756154, 1.570796, 1.683531],accel_mss,speed_ms,0,blend_radius_m)
    movel([0.112369, -1.389479, -2.566941, -0.755968, 1.570796, 1.683166],accel_mss,speed_ms,0,blend_radius_m)
    movel([0.111916, -1.389894, -2.566643, -0.755852, 1.570796, 1.682713],accel_mss,speed_ms,0,blend_radius_m)
    movel([0.111348, -1.390097, -2.566497, -0.755795, 1.570796, 1.682144],accel_mss,speed_ms,0,blend_radius_m)
    movel([0.110638, -1.390114, -2.566485, -0.755790, 1.570796, 1.681434],accel_mss,speed_ms,0,blend_radius_m)
    movel([0.107947, -1.389760, -2.566740, -0.755889, 1.570796, 1.678743],accel_mss,speed_ms,0,blend_radius_m)
    movel([0.105434, -1.389150, -2.567177, -0.756061, 1.570796, 1.676230],accel_mss,speed_ms,0,blend_radius_m)
    movel([0.103104, -1.388299, -2.567788, -0.756302, 1.570796, 1.673901],accel_mss,speed_ms,0,blend_radius_m)
    movel([0.100967, -1.387215, -2.568564, -0.756610, 1.570796, 1.671763],accel_mss,speed_ms,0,blend_radius_m)
    movel([0.099025, -1.385916, -2.569491, -0.756982, 1.570796, 1.669822],accel_mss,speed_ms,0,blend_radius_m)
    movel([0.097291, -1.384409, -2.570564, -0.757416, 1.570796, 1.668087],accel_mss,speed_ms,0,blend_radius_m)
    movel([0.095771, -1.382708, -2.571771, -0.757910, 1.570796, 1.666568],accel_mss,speed_ms,0,blend_radius_m)
    movel([0.094473, -1.380827, -2.573100, -0.758461, 1.570796, 1.665270],accel_mss,speed_ms,0,blend_radius_m)
    movel([0.093411, -1.378773, -2.574547, -0.759069, 1.570796, 1.664208],accel_mss,speed_ms,0,blend_radius_m)
    movel([0.092590, -1.376560, -2.576099, -0.759730, 1.570796, 1.663386],accel_mss,speed_ms,0,blend_radius_m)
    movel([0.092021, -1.374198, -2.577747, -0.760444, 1.570796, 1.662818],accel_mss,speed_ms,0,blend_radius_m)
    movel([0.091719, -1.371698, -2.579483, -0.761208, 1.570796, 1.662515],accel_mss,speed_ms,0,blend_radius_m)
    movel([0.091688, -1.369075, -2.581294, -0.762020, 1.570796, 1.662485],accel_mss,speed_ms,0,blend_radius_m)
    movel([0.091943, -1.366340, -2.583173, -0.762876, 1.570796, 1.662739],accel_mss,speed_ms,0,blend_radius_m)
    movel([0.092496, -1.363503, -2.585110, -0.763775, 1.570796, 1.663292],accel_mss,speed_ms,0,blend_radius_m)
    movel([0.093354, -1.360578, -2.587096, -0.764715, 1.570796, 1.664150],accel_mss,speed_ms,0,blend_radius_m)
    movel([0.095047, -1.356318, -2.589967, -0.766104, 1.570796, 1.665843],accel_mss,speed_ms,0,blend_radius_m)
    movel([0.096067, -1.354205, -2.591381, -0.766803, 1.570796, 1.666864],accel_mss,speed_ms,0,blend_radius_m)
    movel([0.097206, -1.352103, -2.592782, -0.767504, 1.570796, 1.668002],accel_mss,speed_ms,0,blend_radius_m)
    movel([0.098471, -1.350011, -2.594170, -0.768208, 1.570796, 1.669267],accel_mss,speed_ms,0,blend_radius_m)
    movel([0.099865, -1.347930, -2.595545, -0.768914, 1.570796, 1.670662],accel_mss,speed_ms,0,blend_radius_m)
    movel([0.101395, -1.345856, -2.596909, -0.769624, 1.570796, 1.672192],accel_mss,speed_ms,0,blend_radius_m)
    movel([0.103062, -1.343793, -2.598260, -0.770336, 1.570796, 1.673858],accel_mss,speed_ms,0,blend_radius_m)
    movel([0.104534, -1.342128, -2.599346, -0.770915, 1.570796, 1.675330],accel_mss,speed_ms,0,blend_radius_m)
    movel([0.105082, -1.341653, -2.599655, -0.771081, 1.570796, 1.675878],accel_mss,speed_ms,0,blend_radius_m)
    movel([0.105579, -1.341395, -2.599823, -0.771171, 1.570796, 1.676375],accel_mss,speed_ms,0,blend_radius_m)
    movel([0.106077, -1.341339, -2.599860, -0.771190, 1.570796, 1.676873],accel_mss,speed_ms,0,blend_radius_m)
    movel([0.106628, -1.341469, -2.599775, -0.771145, 1.570796, 1.677424],accel_mss,speed_ms,0,blend_radius_m)
    movel([0.108113, -1.342224, -2.599284, -0.770881, 1.570796, 1.678910],accel_mss,speed_ms,0,blend_radius_m)
    movel([0.106316, -1.344176, -2.598009, -0.770203, 1.570796, 1.677112],accel_mss,speed_ms,0,blend_radius_m)
    movel([0.106109, -1.344420, -2.597850, -0.770119, 1.570796, 1.676906],accel_mss,speed_ms,0,blend_radius_m)
    speed_ms = 0.005
    # Splitting Linear movement in 6 (instruction 714: MoveL 662)
    movel([0.106109, -1.342913, -2.597161, -0.772315, 1.570796, 1.676906],accel_mss,speed_ms,0,blend_radius_m)
    movel([0.106109, -1.341410, -2.596471, -0.774508, 1.570796, 1.676906],accel_mss,speed_ms,0,blend_radius_m)
    movel([0.106109, -1.339913, -2.595778, -0.776698, 1.570796, 1.676906],accel_mss,speed_ms,0,blend_radius_m)
    movel([0.106109, -1.338420, -2.595085, -0.778884, 1.570796, 1.676906],accel_mss,speed_ms,0,blend_radius_m)
    movel([0.106109, -1.336932, -2.594389, -0.781068, 1.570796, 1.676906],accel_mss,speed_ms,0,blend_radius_m)
    movel([0.106109, -1.335449, -2.593692, -0.783248, 1.570796, 1.676906],accel_mss,speed_ms,0,blend_radius_m)
    speed_ms = 0.040
    # Splitting Linear movement in 20 (instruction 716: MoveL 663)
    movel([0.106875, -1.333194, -2.595145, -0.784050, 1.570796, 1.677671],accel_mss,speed_ms,0,blend_radius_m)
    movel([0.107644, -1.330931, -2.596596, -0.784862, 1.570796, 1.678441],accel_mss,speed_ms,0,blend_radius_m)
    movel([0.108418, -1.328659, -2.598045, -0.785685, 1.570796, 1.679214],accel_mss,speed_ms,0,blend_radius_m)
    movel([0.109195, -1.326380, -2.599493, -0.786517, 1.570796, 1.679991],accel_mss,speed_ms,0,blend_radius_m)
    movel([0.109976, -1.324091, -2.600939, -0.787359, 1.570796, 1.680773],accel_mss,speed_ms,0,blend_radius_m)
    movel([0.110761, -1.321795, -2.602383, -0.788211, 1.570796, 1.681558],accel_mss,speed_ms,0,blend_radius_m)
    movel([0.111551, -1.319489, -2.603826, -0.789074, 1.570796, 1.682347],accel_mss,speed_ms,0,blend_radius_m)
    movel([0.112344, -1.317175, -2.605267, -0.789947, 1.570796, 1.683140],accel_mss,speed_ms,0,blend_radius_m)
    movel([0.113141, -1.314853, -2.606706, -0.790830, 1.570796, 1.683938],accel_mss,speed_ms,0,blend_radius_m)
    movel([0.113943, -1.312521, -2.608144, -0.791724, 1.570796, 1.684739],accel_mss,speed_ms,0,blend_radius_m)
    movel([0.114748, -1.310181, -2.609580, -0.792628, 1.570796, 1.685545],accel_mss,speed_ms,0,blend_radius_m)
    movel([0.115558, -1.307831, -2.611014, -0.793543, 1.570796, 1.686354],accel_mss,speed_ms,0,blend_radius_m)
    movel([0.116372, -1.305473, -2.612447, -0.794469, 1.570796, 1.687168],accel_mss,speed_ms,0,blend_radius_m)
    movel([0.117190, -1.303106, -2.613878, -0.795405, 1.570796, 1.687987],accel_mss,speed_ms,0,blend_radius_m)
    movel([0.118013, -1.300729, -2.615307, -0.796353, 1.570796, 1.688809],accel_mss,speed_ms,0,blend_radius_m)
    movel([0.118839, -1.298344, -2.616734, -0.797311, 1.570796, 1.689636],accel_mss,speed_ms,0,blend_radius_m)
    movel([0.119671, -1.295949, -2.618160, -0.798281, 1.570796, 1.690467],accel_mss,speed_ms,0,blend_radius_m)
    movel([0.120506, -1.293544, -2.619583, -0.799261, 1.570796, 1.691302],accel_mss,speed_ms,0,blend_radius_m)
    movel([0.121346, -1.291130, -2.621005, -0.800253, 1.570796, 1.692142],accel_mss,speed_ms,0,blend_radius_m)
    movel([0.122190, -1.288707, -2.622426, -0.801257, 1.570796, 1.692987],accel_mss,speed_ms,0,blend_radius_m)
    speed_ms = 0.005
    # Splitting Linear movement in 4 (instruction 718: MoveL 664)
    movel([0.122190, -1.291002, -2.623523, -0.797864, 1.570796, 1.692987],accel_mss,speed_ms,0,blend_radius_m)
    movel([0.122190, -1.293310, -2.624616, -0.794463, 1.570796, 1.692987],accel_mss,speed_ms,0,blend_radius_m)
    movel([0.122190, -1.295630, -2.625706, -0.791053, 1.570796, 1.692987],accel_mss,speed_ms,0,blend_radius_m)
    movel([0.122190, -1.297963, -2.626792, -0.787634, 1.570796, 1.692987],accel_mss,speed_ms,0,blend_radius_m)
    speed_ms = 0.035
    movel([0.121345, -1.299932, -2.625623, -0.786833, 1.570796, 1.692142],accel_mss,speed_ms,0,blend_radius_m)
    movel([0.120728, -1.301794, -2.624514, -0.786081, 1.570796, 1.691524],accel_mss,speed_ms,0,blend_radius_m)
    movel([0.120340, -1.303548, -2.623464, -0.785377, 1.570796, 1.691137],accel_mss,speed_ms,0,blend_radius_m)
    movel([0.120177, -1.305199, -2.622473, -0.784718, 1.570796, 1.690973],accel_mss,speed_ms,0,blend_radius_m)
    movel([0.120238, -1.306748, -2.621539, -0.784102, 1.570796, 1.691034],accel_mss,speed_ms,0,blend_radius_m)
    movel([0.120525, -1.308197, -2.620663, -0.783529, 1.570796, 1.691322],accel_mss,speed_ms,0,blend_radius_m)
    movel([0.121039, -1.309548, -2.619843, -0.782998, 1.570796, 1.691835],accel_mss,speed_ms,0,blend_radius_m)
    movel([0.121775, -1.310804, -2.619079, -0.782506, 1.570796, 1.692571],accel_mss,speed_ms,0,blend_radius_m)
    movel([0.123160, -1.312314, -2.618158, -0.781917, 1.570796, 1.693956],accel_mss,speed_ms,0,blend_radius_m)
    movel([0.124887, -1.313419, -2.617482, -0.781488, 1.570796, 1.695683],accel_mss,speed_ms,0,blend_radius_m)
    movel([0.126906, -1.314127, -2.617048, -0.781214, 1.570796, 1.697702],accel_mss,speed_ms,0,blend_radius_m)
    movel([0.129165, -1.314438, -2.616857, -0.781093, 1.570796, 1.699961],accel_mss,speed_ms,0,blend_radius_m)
    movel([0.131624, -1.314352, -2.616910, -0.781127, 1.570796, 1.702420],accel_mss,speed_ms,0,blend_radius_m)
    movel([0.134231, -1.313872, -2.617205, -0.781313, 1.570796, 1.705027],accel_mss,speed_ms,0,blend_radius_m)
    movel([0.136947, -1.312993, -2.617743, -0.781653, 1.570796, 1.707743],accel_mss,speed_ms,0,blend_radius_m)
    movel([0.139721, -1.311711, -2.618526, -0.782151, 1.570796, 1.710517],accel_mss,speed_ms,0,blend_radius_m)
    movel([0.142427, -1.310077, -2.619521, -0.782790, 1.570796, 1.713223],accel_mss,speed_ms,0,blend_radius_m)
    movel([0.144947, -1.308172, -2.620678, -0.783539, 1.570796, 1.715744],accel_mss,speed_ms,0,blend_radius_m)
    movel([0.147248, -1.306040, -2.621966, -0.784383, 1.570796, 1.718044],accel_mss,speed_ms,0,blend_radius_m)
    movel([0.149284, -1.303726, -2.623357, -0.785306, 1.570796, 1.720081],accel_mss,speed_ms,0,blend_radius_m)
    movel([0.151023, -1.301280, -2.624821, -0.786288, 1.570796, 1.721819],accel_mss,speed_ms,0,blend_radius_m)
    movel([0.152413, -1.298752, -2.626324, -0.787312, 1.570796, 1.723209],accel_mss,speed_ms,0,blend_radius_m)
    movel([0.153421, -1.296189, -2.627841, -0.788359, 1.570796, 1.724218],accel_mss,speed_ms,0,blend_radius_m)
    movel([0.153997, -1.293642, -2.629339, -0.789407, 1.570796, 1.724793],accel_mss,speed_ms,0,blend_radius_m)
    movel([0.154134, -1.291082, -2.630837, -0.790469, 1.570796, 1.724930],accel_mss,speed_ms,0,blend_radius_m)
    movel([0.153815, -1.288798, -2.632167, -0.791424, 1.570796, 1.724612],accel_mss,speed_ms,0,blend_radius_m)
    movel([0.153057, -1.286822, -2.633311, -0.792255, 1.570796, 1.723854],accel_mss,speed_ms,0,blend_radius_m)
    movel([0.151885, -1.285181, -2.634258, -0.792949, 1.570796, 1.722682],accel_mss,speed_ms,0,blend_radius_m)
    movel([0.150315, -1.283903, -2.634993, -0.793492, 1.570796, 1.721111],accel_mss,speed_ms,0,blend_radius_m)
    movel([0.148371, -1.283016, -2.635502, -0.793870, 1.570796, 1.719168],accel_mss,speed_ms,0,blend_radius_m)
    movel([0.146077, -1.282549, -2.635770, -0.794070, 1.570796, 1.716873],accel_mss,speed_ms,0,blend_radius_m)
    movel([0.143454, -1.282525, -2.635784, -0.794080, 1.570796, 1.714250],accel_mss,speed_ms,0,blend_radius_m)
    movel([0.141686, -1.282809, -2.635621, -0.793959, 1.570796, 1.712483],accel_mss,speed_ms,0,blend_radius_m)
    movel([0.141035, -1.283059, -2.635478, -0.793852, 1.570796, 1.711832],accel_mss,speed_ms,0,blend_radius_m)
    movel([0.140530, -1.283391, -2.635287, -0.793711, 1.570796, 1.711326],accel_mss,speed_ms,0,blend_radius_m)
    movel([0.140166, -1.283807, -2.635048, -0.793533, 1.570796, 1.710962],accel_mss,speed_ms,0,blend_radius_m)
    movel([0.139936, -1.284321, -2.634753, -0.793315, 1.570796, 1.710733],accel_mss,speed_ms,0,blend_radius_m)
    movel([0.139857, -1.285655, -2.633985, -0.792749, 1.570796, 1.710654],accel_mss,speed_ms,0,blend_radius_m)
    movel([0.140062, -1.286014, -2.633778, -0.792597, 1.570796, 1.710859],accel_mss,speed_ms,0,blend_radius_m)
    movel([0.140512, -1.286275, -2.633628, -0.792487, 1.570796, 1.711308],accel_mss,speed_ms,0,blend_radius_m)
    movel([0.141094, -1.286419, -2.633545, -0.792426, 1.570796, 1.711890],accel_mss,speed_ms,0,blend_radius_m)
    movel([0.143913, -1.286469, -2.633515, -0.792404, 1.570796, 1.714709],accel_mss,speed_ms,0,blend_radius_m)
    movel([0.145854, -1.286942, -2.633242, -0.792205, 1.570796, 1.716650],accel_mss,speed_ms,0,blend_radius_m)
    movel([0.147474, -1.287813, -2.632738, -0.791838, 1.570796, 1.718271],accel_mss,speed_ms,0,blend_radius_m)
    movel([0.148747, -1.289036, -2.632029, -0.791324, 1.570796, 1.719543],accel_mss,speed_ms,0,blend_radius_m)
    movel([0.149631, -1.290566, -2.631138, -0.790684, 1.570796, 1.720427],accel_mss,speed_ms,0,blend_radius_m)
    movel([0.150095, -1.292360, -2.630091, -0.789938, 1.570796, 1.720892],accel_mss,speed_ms,0,blend_radius_m)
    movel([0.150108, -1.294370, -2.628912, -0.789107, 1.570796, 1.720905],accel_mss,speed_ms,0,blend_radius_m)
    movel([0.149938, -1.295443, -2.628281, -0.788665, 1.570796, 1.720734],accel_mss,speed_ms,0,blend_radius_m)
    movel([0.149201, -1.297760, -2.626912, -0.787716, 1.570796, 1.719997],accel_mss,speed_ms,0,blend_radius_m)
    movel([0.148659, -1.298949, -2.626208, -0.787232, 1.570796, 1.719455],accel_mss,speed_ms,0,blend_radius_m)
    movel([0.147296, -1.301249, -2.624839, -0.786301, 1.570796, 1.718093],accel_mss,speed_ms,0,blend_radius_m)
    movel([0.145613, -1.303404, -2.623550, -0.785435, 1.570796, 1.716410],accel_mss,speed_ms,0,blend_radius_m)
    movel([0.143668, -1.305367, -2.622371, -0.784651, 1.570796, 1.714464],accel_mss,speed_ms,0,blend_radius_m)
    movel([0.141512, -1.307092, -2.621331, -0.783966, 1.570796, 1.712308],accel_mss,speed_ms,0,blend_radius_m)
    movel([0.139201, -1.308533, -2.620459, -0.783397, 1.570796, 1.709997],accel_mss,speed_ms,0,blend_radius_m)
    movel([0.136788, -1.309640, -2.619788, -0.782962, 1.570796, 1.707584],accel_mss,speed_ms,0,blend_radius_m)
    movel([0.135561, -1.310054, -2.619536, -0.782799, 1.570796, 1.706357],accel_mss,speed_ms,0,blend_radius_m)
    movel([0.134326, -1.310370, -2.619344, -0.782676, 1.570796, 1.705123],accel_mss,speed_ms,0,blend_radius_m)
    movel([0.131994, -1.310660, -2.619167, -0.782562, 1.570796, 1.702791],accel_mss,speed_ms,0,blend_radius_m)
    movel([0.129883, -1.310520, -2.619252, -0.782617, 1.570796, 1.700680],accel_mss,speed_ms,0,blend_radius_m)
    movel([0.128042, -1.309974, -2.619584, -0.782831, 1.570796, 1.698839],accel_mss,speed_ms,0,blend_radius_m)
    movel([0.126514, -1.309054, -2.620143, -0.783192, 1.570796, 1.697310],accel_mss,speed_ms,0,blend_radius_m)
    movel([0.125344, -1.307792, -2.620908, -0.783689, 1.570796, 1.696140],accel_mss,speed_ms,0,blend_radius_m)
    movel([0.124583, -1.306207, -2.621865, -0.784317, 1.570796, 1.695379],accel_mss,speed_ms,0,blend_radius_m)
    movel([0.124369, -1.305304, -2.622409, -0.784676, 1.570796, 1.695165],accel_mss,speed_ms,0,blend_radius_m)
    movel([0.124274, -1.304334, -2.622992, -0.785063, 1.570796, 1.695070],accel_mss,speed_ms,0,blend_radius_m)
    movel([0.124471, -1.302193, -2.624275, -0.785921, 1.570796, 1.695267],accel_mss,speed_ms,0,blend_radius_m)
    movel([0.124610, -1.300631, -2.625207, -0.786550, 1.570796, 1.695406],accel_mss,speed_ms,0,blend_radius_m)
    movel([0.124287, -1.299454, -2.625908, -0.787027, 1.570796, 1.695083],accel_mss,speed_ms,0,blend_radius_m)
    movel([0.123483, -1.298589, -2.626421, -0.787379, 1.570796, 1.694280],accel_mss,speed_ms,0,blend_radius_m)
    movel([0.122190, -1.297963, -2.626792, -0.787634, 1.570796, 1.692987],accel_mss,speed_ms,0,blend_radius_m)
    movel([0.121345, -1.299932, -2.625623, -0.786833, 1.570796, 1.692142],accel_mss,speed_ms,0,blend_radius_m)
    movel([0.121138, -1.300559, -2.625250, -0.786580, 1.570796, 1.691935],accel_mss,speed_ms,0,blend_radius_m)
    speed_ms = 0.005
    # Splitting Linear movement in 4 (instruction 795: MoveL 739)
    movel([0.121138, -1.298230, -2.624167, -0.789992, 1.570796, 1.691935],accel_mss,speed_ms,0,blend_radius_m)
    movel([0.121138, -1.295914, -2.623080, -0.793395, 1.570796, 1.691935],accel_mss,speed_ms,0,blend_radius_m)
    movel([0.121138, -1.293609, -2.621989, -0.796790, 1.570796, 1.691935],accel_mss,speed_ms,0,blend_radius_m)
    movel([0.121138, -1.291318, -2.620895, -0.800176, 1.570796, 1.691935],accel_mss,speed_ms,0,blend_radius_m)
    speed_ms = 0.040
    # Splitting Linear movement in 10 (instruction 797: MoveL 740)
    movel([0.120168, -1.289572, -2.621919, -0.800898, 1.570796, 1.690965],accel_mss,speed_ms,0,blend_radius_m)
    movel([0.119193, -1.287825, -2.622940, -0.801624, 1.570796, 1.689990],accel_mss,speed_ms,0,blend_radius_m)
    movel([0.118214, -1.286077, -2.623958, -0.802354, 1.570796, 1.689011],accel_mss,speed_ms,0,blend_radius_m)
    movel([0.117231, -1.284326, -2.624974, -0.803089, 1.570796, 1.688027],accel_mss,speed_ms,0,blend_radius_m)
    movel([0.116242, -1.282574, -2.625986, -0.803829, 1.570796, 1.687039],accel_mss,speed_ms,0,blend_radius_m)
    movel([0.115250, -1.280820, -2.626995, -0.804573, 1.570796, 1.686046],accel_mss,speed_ms,0,blend_radius_m)
    movel([0.114252, -1.279065, -2.628002, -0.805322, 1.570796, 1.685049],accel_mss,speed_ms,0,blend_radius_m)
    movel([0.113250, -1.277308, -2.629006, -0.806076, 1.570796, 1.684047],accel_mss,speed_ms,0,blend_radius_m)
    movel([0.112244, -1.275549, -2.630006, -0.806833, 1.570796, 1.683040],accel_mss,speed_ms,0,blend_radius_m)
    movel([0.111232, -1.273789, -2.631004, -0.807596, 1.570796, 1.682029],accel_mss,speed_ms,0,blend_radius_m)
    speed_ms = 0.005
    # Splitting Linear movement in 6 (instruction 799: MoveL 741)
    movel([0.111232, -1.275331, -2.631747, -0.805311, 1.570796, 1.682029],accel_mss,speed_ms,0,blend_radius_m)
    movel([0.111232, -1.276879, -2.632489, -0.803021, 1.570796, 1.682029],accel_mss,speed_ms,0,blend_radius_m)
    movel([0.111232, -1.278433, -2.633228, -0.800728, 1.570796, 1.682029],accel_mss,speed_ms,0,blend_radius_m)
    movel([0.111232, -1.279992, -2.633967, -0.798430, 1.570796, 1.682029],accel_mss,speed_ms,0,blend_radius_m)
    movel([0.111232, -1.281557, -2.634703, -0.796129, 1.570796, 1.682029],accel_mss,speed_ms,0,blend_radius_m)
    movel([0.111232, -1.283128, -2.635438, -0.793823, 1.570796, 1.682029],accel_mss,speed_ms,0,blend_radius_m)
    speed_ms = 0.035
    movel([0.108593, -1.286019, -2.633775, -0.792595, 1.570796, 1.679389],accel_mss,speed_ms,0,blend_radius_m)
    movel([0.106209, -1.289014, -2.632042, -0.791334, 1.570796, 1.677005],accel_mss,speed_ms,0,blend_radius_m)
    movel([0.104085, -1.292083, -2.630253, -0.790053, 1.570796, 1.674882],accel_mss,speed_ms,0,blend_radius_m)
    movel([0.102227, -1.295203, -2.628422, -0.788764, 1.570796, 1.673023],accel_mss,speed_ms,0,blend_radius_m)
    movel([0.100631, -1.298351, -2.626563, -0.787476, 1.570796, 1.671427],accel_mss,speed_ms,0,blend_radius_m)
    movel([0.099307, -1.301496, -2.624692, -0.786201, 1.570796, 1.670103],accel_mss,speed_ms,0,blend_radius_m)
    movel([0.098254, -1.304622, -2.622819, -0.784948, 1.570796, 1.669050],accel_mss,speed_ms,0,blend_radius_m)
    movel([0.097473, -1.307701, -2.620963, -0.783725, 1.570796, 1.668269],accel_mss,speed_ms,0,blend_radius_m)
    movel([0.096969, -1.310714, -2.619134, -0.782541, 1.570796, 1.667765],accel_mss,speed_ms,0,blend_radius_m)
    movel([0.096738, -1.313642, -2.617346, -0.781402, 1.570796, 1.667534],accel_mss,speed_ms,0,blend_radius_m)
    movel([0.096788, -1.316458, -2.615615, -0.780316, 1.570796, 1.667584],accel_mss,speed_ms,0,blend_radius_m)
    movel([0.097117, -1.319148, -2.613951, -0.779290, 1.570796, 1.667913],accel_mss,speed_ms,0,blend_radius_m)
    movel([0.097729, -1.321687, -2.612373, -0.778330, 1.570796, 1.668525],accel_mss,speed_ms,0,blend_radius_m)
    movel([0.098624, -1.324055, -2.610892, -0.777441, 1.570796, 1.669421],accel_mss,speed_ms,0,blend_radius_m)
    movel([0.099806, -1.326238, -2.609521, -0.776630, 1.570796, 1.670603],accel_mss,speed_ms,0,blend_radius_m)
    movel([0.101278, -1.328214, -2.608274, -0.775900, 1.570796, 1.672074],accel_mss,speed_ms,0,blend_radius_m)
    movel([0.103099, -1.330034, -2.607122, -0.775233, 1.570796, 1.673895],accel_mss,speed_ms,0,blend_radius_m)
    movel([0.105155, -1.331578, -2.606140, -0.774671, 1.570796, 1.675952],accel_mss,speed_ms,0,blend_radius_m)
    movel([0.107423, -1.332852, -2.605328, -0.774209, 1.570796, 1.678219],accel_mss,speed_ms,0,blend_radius_m)
    movel([0.109886, -1.333860, -2.604684, -0.773846, 1.570796, 1.680682],accel_mss,speed_ms,0,blend_radius_m)
    movel([0.112523, -1.334603, -2.604207, -0.773578, 1.570796, 1.683319],accel_mss,speed_ms,0,blend_radius_m)
    movel([0.115317, -1.335085, -2.603898, -0.773405, 1.570796, 1.686113],accel_mss,speed_ms,0,blend_radius_m)
    movel([0.118243, -1.335309, -2.603754, -0.773325, 1.570796, 1.689040],accel_mss,speed_ms,0,blend_radius_m)
    movel([0.121288, -1.335277, -2.603775, -0.773337, 1.570796, 1.692084],accel_mss,speed_ms,0,blend_radius_m)
    movel([0.124434, -1.334985, -2.603962, -0.773441, 1.570796, 1.695230],accel_mss,speed_ms,0,blend_radius_m)
    movel([0.127659, -1.334440, -2.604312, -0.773637, 1.570796, 1.698455],accel_mss,speed_ms,0,blend_radius_m)
    movel([0.130948, -1.333640, -2.604824, -0.773925, 1.570796, 1.701744],accel_mss,speed_ms,0,blend_radius_m)
    movel([0.134283, -1.332580, -2.605501, -0.774307, 1.570796, 1.705080],accel_mss,speed_ms,0,blend_radius_m)
    movel([0.137648, -1.331265, -2.606339, -0.774785, 1.570796, 1.708444],accel_mss,speed_ms,0,blend_radius_m)
    movel([0.141024, -1.329690, -2.607340, -0.775359, 1.570796, 1.711820],accel_mss,speed_ms,0,blend_radius_m)
    movel([0.144395, -1.327850, -2.608504, -0.776034, 1.570796, 1.715191],accel_mss,speed_ms,0,blend_radius_m)
    movel([0.147741, -1.325748, -2.609830, -0.776811, 1.570796, 1.718537],accel_mss,speed_ms,0,blend_radius_m)
    movel([0.151168, -1.323307, -2.611361, -0.777721, 1.570796, 1.721964],accel_mss,speed_ms,0,blend_radius_m)
    movel([0.154411, -1.320709, -2.612982, -0.778698, 1.570796, 1.725207],accel_mss,speed_ms,0,blend_radius_m)
    movel([0.157467, -1.317973, -2.614679, -0.779737, 1.570796, 1.728264],accel_mss,speed_ms,0,blend_radius_m)
    movel([0.160325, -1.315107, -2.616446, -0.780836, 1.570796, 1.731121],accel_mss,speed_ms,0,blend_radius_m)
    movel([0.162972, -1.312131, -2.618270, -0.781988, 1.570796, 1.733769],accel_mss,speed_ms,0,blend_radius_m)
    movel([0.165403, -1.309057, -2.620141, -0.783191, 1.570796, 1.736199],accel_mss,speed_ms,0,blend_radius_m)
    movel([0.167601, -1.305901, -2.622050, -0.784438, 1.570796, 1.738397],accel_mss,speed_ms,0,blend_radius_m)
    movel([0.169559, -1.302682, -2.623983, -0.785724, 1.570796, 1.740356],accel_mss,speed_ms,0,blend_radius_m)
    movel([0.171264, -1.299416, -2.625931, -0.787043, 1.570796, 1.742060],accel_mss,speed_ms,0,blend_radius_m)
    movel([0.172702, -1.296116, -2.627884, -0.788389, 1.570796, 1.743498],accel_mss,speed_ms,0,blend_radius_m)
    movel([0.173861, -1.292807, -2.629829, -0.789753, 1.570796, 1.744657],accel_mss,speed_ms,0,blend_radius_m)
    movel([0.174729, -1.289503, -2.631757, -0.791129, 1.570796, 1.745525],accel_mss,speed_ms,0,blend_radius_m)
    movel([0.175291, -1.286223, -2.633657, -0.792508, 1.570796, 1.746087],accel_mss,speed_ms,0,blend_radius_m)
    movel([0.175532, -1.282991, -2.635517, -0.793881, 1.570796, 1.746328],accel_mss,speed_ms,0,blend_radius_m)
    movel([0.175444, -1.279825, -2.637325, -0.795239, 1.570796, 1.746240],accel_mss,speed_ms,0,blend_radius_m)
    movel([0.175005, -1.276747, -2.639071, -0.796571, 1.570796, 1.745801],accel_mss,speed_ms,0,blend_radius_m)
    movel([0.174329, -1.274254, -2.640477, -0.797658, 1.570796, 1.745126],accel_mss,speed_ms,0,blend_radius_m)
    movel([0.173383, -1.271971, -2.641757, -0.798661, 1.570796, 1.744180],accel_mss,speed_ms,0,blend_radius_m)
    movel([0.172181, -1.269906, -2.642910, -0.799574, 1.570796, 1.742977],accel_mss,speed_ms,0,blend_radius_m)
    movel([0.170744, -1.268054, -2.643939, -0.800396, 1.570796, 1.741540],accel_mss,speed_ms,0,blend_radius_m)
    movel([0.169097, -1.266418, -2.644844, -0.801127, 1.570796, 1.739893],accel_mss,speed_ms,0,blend_radius_m)
    movel([0.167259, -1.265005, -2.645624, -0.801760, 1.570796, 1.738056],accel_mss,speed_ms,0,blend_radius_m)
    movel([0.165253, -1.263811, -2.646281, -0.802297, 1.570796, 1.736049],accel_mss,speed_ms,0,blend_radius_m)
    movel([0.163103, -1.262839, -2.646814, -0.802736, 1.570796, 1.733899],accel_mss,speed_ms,0,blend_radius_m)
    movel([0.160832, -1.262085, -2.647227, -0.803077, 1.570796, 1.731628],accel_mss,speed_ms,0,blend_radius_m)
    movel([0.158462, -1.261555, -2.647517, -0.803317, 1.570796, 1.729259],accel_mss,speed_ms,0,blend_radius_m)
    movel([0.156018, -1.261242, -2.647688, -0.803459, 1.570796, 1.726815],accel_mss,speed_ms,0,blend_radius_m)
    movel([0.153526, -1.261146, -2.647740, -0.803503, 1.570796, 1.724323],accel_mss,speed_ms,0,blend_radius_m)
    movel([0.151007, -1.261266, -2.647675, -0.803448, 1.570796, 1.721803],accel_mss,speed_ms,0,blend_radius_m)
    movel([0.148489, -1.261602, -2.647491, -0.803296, 1.570796, 1.719285],accel_mss,speed_ms,0,blend_radius_m)
    movel([0.145992, -1.262145, -2.647194, -0.803050, 1.570796, 1.716788],accel_mss,speed_ms,0,blend_radius_m)
    movel([0.143542, -1.262898, -2.646781, -0.802709, 1.570796, 1.714338],accel_mss,speed_ms,0,blend_radius_m)
    movel([0.142953, -1.264867, -2.645700, -0.801822, 1.570796, 1.713750],accel_mss,speed_ms,0,blend_radius_m)
    movel([0.142872, -1.265473, -2.645366, -0.801550, 1.570796, 1.713668],accel_mss,speed_ms,0,blend_radius_m)
    movel([0.142954, -1.265865, -2.645149, -0.801374, 1.570796, 1.713750],accel_mss,speed_ms,0,blend_radius_m)
    movel([0.143214, -1.266079, -2.645031, -0.801278, 1.570796, 1.714011],accel_mss,speed_ms,0,blend_radius_m)
    movel([0.143675, -1.266137, -2.644999, -0.801252, 1.570796, 1.714472],accel_mss,speed_ms,0,blend_radius_m)
    movel([0.148316, -1.265486, -2.645359, -0.801544, 1.570796, 1.719112],accel_mss,speed_ms,0,blend_radius_m)
    movel([0.151240, -1.265323, -2.645449, -0.801618, 1.570796, 1.722037],accel_mss,speed_ms,0,blend_radius_m)
    movel([0.154010, -1.265422, -2.645394, -0.801573, 1.570796, 1.724806],accel_mss,speed_ms,0,blend_radius_m)
    movel([0.156618, -1.265781, -2.645196, -0.801412, 1.570796, 1.727415],accel_mss,speed_ms,0,blend_radius_m)
    movel([0.159047, -1.266388, -2.644861, -0.801140, 1.570796, 1.729843],accel_mss,speed_ms,0,blend_radius_m)
    movel([0.161290, -1.267233, -2.644393, -0.800762, 1.570796, 1.732086],accel_mss,speed_ms,0,blend_radius_m)
    movel([0.163333, -1.268309, -2.643797, -0.800283, 1.570796, 1.734129],accel_mss,speed_ms,0,blend_radius_m)
    movel([0.165170, -1.269605, -2.643077, -0.799707, 1.570796, 1.735967],accel_mss,speed_ms,0,blend_radius_m)
    movel([0.166792, -1.271110, -2.642238, -0.799041, 1.570796, 1.737588],accel_mss,speed_ms,0,blend_radius_m)
    movel([0.168184, -1.272817, -2.641283, -0.798288, 1.570796, 1.738981],accel_mss,speed_ms,0,blend_radius_m)
    movel([0.169340, -1.274712, -2.640219, -0.797458, 1.570796, 1.740137],accel_mss,speed_ms,0,blend_radius_m)
    movel([0.170255, -1.276785, -2.639049, -0.796554, 1.570796, 1.741051],accel_mss,speed_ms,0,blend_radius_m)
    movel([0.170920, -1.279025, -2.637780, -0.795584, 1.570796, 1.741716],accel_mss,speed_ms,0,blend_radius_m)
    movel([0.171322, -1.281423, -2.636414, -0.794552, 1.570796, 1.742118],accel_mss,speed_ms,0,blend_radius_m)
    movel([0.171458, -1.283968, -2.634956, -0.793465, 1.570796, 1.742254],accel_mss,speed_ms,0,blend_radius_m)
    movel([0.171323, -1.286650, -2.633411, -0.792328, 1.570796, 1.742119],accel_mss,speed_ms,0,blend_radius_m)
    movel([0.170903, -1.289513, -2.631752, -0.791125, 1.570796, 1.741699],accel_mss,speed_ms,0,blend_radius_m)
    movel([0.170233, -1.292385, -2.630076, -0.789928, 1.570796, 1.741029],accel_mss,speed_ms,0,blend_radius_m)
    movel([0.169320, -1.295255, -2.628392, -0.788743, 1.570796, 1.740116],accel_mss,speed_ms,0,blend_radius_m)
    movel([0.168181, -1.298105, -2.626708, -0.787576, 1.570796, 1.738977],accel_mss,speed_ms,0,blend_radius_m)
    movel([0.166826, -1.300926, -2.625032, -0.786432, 1.570796, 1.737623],accel_mss,speed_ms,0,blend_radius_m)
    movel([0.165266, -1.303700, -2.623373, -0.785316, 1.570796, 1.736062],accel_mss,speed_ms,0,blend_radius_m)
    movel([0.163518, -1.306416, -2.621739, -0.784234, 1.570796, 1.734314],accel_mss,speed_ms,0,blend_radius_m)
    movel([0.161587, -1.309062, -2.620138, -0.783189, 1.570796, 1.732383],accel_mss,speed_ms,0,blend_radius_m)
    movel([0.159488, -1.311625, -2.618579, -0.782185, 1.570796, 1.730285],accel_mss,speed_ms,0,blend_radius_m)
    movel([0.157233, -1.314095, -2.617068, -0.781226, 1.570796, 1.728029],accel_mss,speed_ms,0,blend_radius_m)
    movel([0.154830, -1.316462, -2.615612, -0.780315, 1.570796, 1.725626],accel_mss,speed_ms,0,blend_radius_m)
    movel([0.152288, -1.318709, -2.614224, -0.779457, 1.570796, 1.723084],accel_mss,speed_ms,0,blend_radius_m)
    movel([0.149618, -1.320828, -2.612908, -0.778653, 1.570796, 1.720415],accel_mss,speed_ms,0,blend_radius_m)
    movel([0.146830, -1.322810, -2.611671, -0.777907, 1.570796, 1.717627],accel_mss,speed_ms,0,blend_radius_m)
    movel([0.143935, -1.324643, -2.610524, -0.777222, 1.570796, 1.714732],accel_mss,speed_ms,0,blend_radius_m)
    movel([0.140937, -1.326314, -2.609473, -0.776601, 1.570796, 1.711733],accel_mss,speed_ms,0,blend_radius_m)
    movel([0.138227, -1.327636, -2.608640, -0.776113, 1.570796, 1.709024],accel_mss,speed_ms,0,blend_radius_m)
    movel([0.135534, -1.328773, -2.607921, -0.775695, 1.570796, 1.706330],accel_mss,speed_ms,0,blend_radius_m)
    movel([0.132865, -1.329720, -2.607321, -0.775348, 1.570796, 1.703661],accel_mss,speed_ms,0,blend_radius_m)
    movel([0.130234, -1.330486, -2.606835, -0.775068, 1.570796, 1.701030],accel_mss,speed_ms,0,blend_radius_m)
    movel([0.127647, -1.331067, -2.606465, -0.774857, 1.570796, 1.698443],accel_mss,speed_ms,0,blend_radius_m)
    movel([0.125117, -1.331468, -2.606210, -0.774711, 1.570796, 1.695913],accel_mss,speed_ms,0,blend_radius_m)
    movel([0.122651, -1.331685, -2.606072, -0.774632, 1.570796, 1.693448],accel_mss,speed_ms,0,blend_radius_m)
    movel([0.120258, -1.331724, -2.606047, -0.774618, 1.570796, 1.691054],accel_mss,speed_ms,0,blend_radius_m)
    movel([0.117950, -1.331583, -2.606137, -0.774669, 1.570796, 1.688747],accel_mss,speed_ms,0,blend_radius_m)
    movel([0.115738, -1.331260, -2.606342, -0.774786, 1.570796, 1.686534],accel_mss,speed_ms,0,blend_radius_m)
    movel([0.113627, -1.330760, -2.606661, -0.774969, 1.570796, 1.684424],accel_mss,speed_ms,0,blend_radius_m)
    movel([0.111633, -1.330077, -2.607095, -0.775218, 1.570796, 1.682430],accel_mss,speed_ms,0,blend_radius_m)
    movel([0.109765, -1.329213, -2.607643, -0.775534, 1.570796, 1.680561],accel_mss,speed_ms,0,blend_radius_m)
    movel([0.108035, -1.328164, -2.608306, -0.775919, 1.570796, 1.678831],accel_mss,speed_ms,0,blend_radius_m)
    movel([0.106450, -1.326936, -2.609082, -0.776372, 1.570796, 1.677246],accel_mss,speed_ms,0,blend_radius_m)
    movel([0.105024, -1.325520, -2.609973, -0.776896, 1.570796, 1.675820],accel_mss,speed_ms,0,blend_radius_m)
    movel([0.103789, -1.323943, -2.610962, -0.777483, 1.570796, 1.674585],accel_mss,speed_ms,0,blend_radius_m)
    movel([0.102760, -1.322228, -2.612035, -0.778126, 1.570796, 1.673556],accel_mss,speed_ms,0,blend_radius_m)
    movel([0.101937, -1.320387, -2.613182, -0.778820, 1.570796, 1.672734],accel_mss,speed_ms,0,blend_radius_m)
    movel([0.101320, -1.318424, -2.614400, -0.779565, 1.570796, 1.672116],accel_mss,speed_ms,0,blend_radius_m)
    movel([0.100909, -1.316353, -2.615679, -0.780357, 1.570796, 1.671706],accel_mss,speed_ms,0,blend_radius_m)
    movel([0.100706, -1.314183, -2.617014, -0.781192, 1.570796, 1.671503],accel_mss,speed_ms,0,blend_radius_m)
    movel([0.100706, -1.311923, -2.618397, -0.782069, 1.570796, 1.671502],accel_mss,speed_ms,0,blend_radius_m)
    movel([0.100914, -1.309581, -2.619823, -0.782985, 1.570796, 1.671710],accel_mss,speed_ms,0,blend_radius_m)
    movel([0.101330, -1.307172, -2.621283, -0.783934, 1.570796, 1.672126],accel_mss,speed_ms,0,blend_radius_m)
    movel([0.101950, -1.304703, -2.622771, -0.784915, 1.570796, 1.672746],accel_mss,speed_ms,0,blend_radius_m)
    movel([0.102777, -1.302185, -2.624280, -0.785924, 1.570796, 1.673573],accel_mss,speed_ms,0,blend_radius_m)
    movel([0.103813, -1.299626, -2.625806, -0.786958, 1.570796, 1.674610],accel_mss,speed_ms,0,blend_radius_m)
    movel([0.105054, -1.297044, -2.627336, -0.788009, 1.570796, 1.675850],accel_mss,speed_ms,0,blend_radius_m)
    movel([0.106503, -1.294446, -2.628868, -0.789075, 1.570796, 1.677299],accel_mss,speed_ms,0,blend_radius_m)
    movel([0.108159, -1.291844, -2.630393, -0.790152, 1.570796, 1.678955],accel_mss,speed_ms,0,blend_radius_m)
    movel([0.110023, -1.289251, -2.631904, -0.791234, 1.570796, 1.680819],accel_mss,speed_ms,0,blend_radius_m)
    movel([0.113606, -1.284674, -2.634550, -0.793165, 1.570796, 1.684402],accel_mss,speed_ms,0,blend_radius_m)
    movel([0.112390, -1.283747, -2.635083, -0.793559, 1.570796, 1.683186],accel_mss,speed_ms,0,blend_radius_m)
    movel([0.111232, -1.283128, -2.635438, -0.793823, 1.570796, 1.682029],accel_mss,speed_ms,0,blend_radius_m)
    movel([0.109028, -1.285544, -2.634049, -0.792796, 1.570796, 1.679824],accel_mss,speed_ms,0,blend_radius_m)
    speed_ms = 0.005
    # Splitting Linear movement in 4 (instruction 939: MoveL 879)
    movel([0.109028, -1.283193, -2.632949, -0.796247, 1.570796, 1.679824],accel_mss,speed_ms,0,blend_radius_m)
    movel([0.109028, -1.280855, -2.631845, -0.799689, 1.570796, 1.679824],accel_mss,speed_ms,0,blend_radius_m)
    movel([0.109028, -1.278530, -2.630738, -0.803121, 1.570796, 1.679824],accel_mss,speed_ms,0,blend_radius_m)
    movel([0.109028, -1.276218, -2.629626, -0.806545, 1.570796, 1.679824],accel_mss,speed_ms,0,blend_radius_m)
    speed_ms = 0.040
    # Splitting Linear movement in 24 (instruction 941: MoveL 880)
    movel([0.111193, -1.273943, -2.630917, -0.807529, 1.570796, 1.681990],accel_mss,speed_ms,0,blend_radius_m)
    movel([0.113368, -1.271660, -2.632206, -0.808523, 1.570796, 1.684164],accel_mss,speed_ms,0,blend_radius_m)
    movel([0.115552, -1.269370, -2.633492, -0.809527, 1.570796, 1.686348],accel_mss,speed_ms,0,blend_radius_m)
    movel([0.117745, -1.267072, -2.634776, -0.810540, 1.570796, 1.688542],accel_mss,speed_ms,0,blend_radius_m)
    movel([0.119948, -1.264768, -2.636058, -0.811564, 1.570796, 1.690744],accel_mss,speed_ms,0,blend_radius_m)
    movel([0.122160, -1.262455, -2.637337, -0.812597, 1.570796, 1.692957],accel_mss,speed_ms,0,blend_radius_m)
    movel([0.124382, -1.260135, -2.638614, -0.813639, 1.570796, 1.695179],accel_mss,speed_ms,0,blend_radius_m)
    movel([0.126614, -1.257808, -2.639888, -0.814692, 1.570796, 1.697410],accel_mss,speed_ms,0,blend_radius_m)
    movel([0.128855, -1.255473, -2.641161, -0.815755, 1.570796, 1.699651],accel_mss,speed_ms,0,blend_radius_m)
    movel([0.131106, -1.253131, -2.642430, -0.816828, 1.570796, 1.701902],accel_mss,speed_ms,0,blend_radius_m)
    movel([0.133367, -1.250780, -2.643697, -0.817911, 1.570796, 1.704163],accel_mss,speed_ms,0,blend_radius_m)
    movel([0.135637, -1.248422, -2.644962, -0.819005, 1.570796, 1.706433],accel_mss,speed_ms,0,blend_radius_m)
    movel([0.137917, -1.246056, -2.646225, -0.820108, 1.570796, 1.708714],accel_mss,speed_ms,0,blend_radius_m)
    movel([0.140208, -1.243683, -2.647484, -0.821222, 1.570796, 1.711004],accel_mss,speed_ms,0,blend_radius_m)
    movel([0.142508, -1.241301, -2.648742, -0.822346, 1.570796, 1.713304],accel_mss,speed_ms,0,blend_radius_m)
    movel([0.144818, -1.238911, -2.649996, -0.823481, 1.570796, 1.715615],accel_mss,speed_ms,0,blend_radius_m)
    movel([0.147139, -1.236514, -2.651249, -0.824626, 1.570796, 1.717935],accel_mss,speed_ms,0,blend_radius_m)
    movel([0.149470, -1.234108, -2.652499, -0.825782, 1.570796, 1.720266],accel_mss,speed_ms,0,blend_radius_m)
    movel([0.151811, -1.231695, -2.653746, -0.826949, 1.570796, 1.722607],accel_mss,speed_ms,0,blend_radius_m)
    movel([0.154162, -1.229273, -2.654990, -0.828126, 1.570796, 1.724958],accel_mss,speed_ms,0,blend_radius_m)
    movel([0.156523, -1.226843, -2.656232, -0.829314, 1.570796, 1.727320],accel_mss,speed_ms,0,blend_radius_m)
    movel([0.158895, -1.224405, -2.657472, -0.830513, 1.570796, 1.729692],accel_mss,speed_ms,0,blend_radius_m)
    movel([0.161278, -1.221958, -2.658708, -0.831723, 1.570796, 1.732074],accel_mss,speed_ms,0,blend_radius_m)
    movel([0.163671, -1.219503, -2.659943, -0.832943, 1.570796, 1.734467],accel_mss,speed_ms,0,blend_radius_m)
    speed_ms = 0.005
    # Splitting Linear movement in 6 (instruction 943: MoveL 881)
    movel([0.163671, -1.221087, -2.660727, -0.830576, 1.570796, 1.734467],accel_mss,speed_ms,0,blend_radius_m)
    movel([0.163671, -1.222677, -2.661509, -0.828203, 1.570796, 1.734467],accel_mss,speed_ms,0,blend_radius_m)
    movel([0.163671, -1.224273, -2.662290, -0.825826, 1.570796, 1.734467],accel_mss,speed_ms,0,blend_radius_m)
    movel([0.163671, -1.225876, -2.663069, -0.823444, 1.570796, 1.734467],accel_mss,speed_ms,0,blend_radius_m)
    movel([0.163671, -1.227486, -2.663847, -0.821056, 1.570796, 1.734467],accel_mss,speed_ms,0,blend_radius_m)
    movel([0.163671, -1.229102, -2.664623, -0.818664, 1.570796, 1.734467],accel_mss,speed_ms,0,blend_radius_m)
    speed_ms = 0.035
    movel([0.165524, -1.226318, -2.666033, -0.820038, 1.570796, 1.736320],accel_mss,speed_ms,0,blend_radius_m)
    movel([0.166959, -1.223449, -2.667476, -0.821464, 1.570796, 1.737756],accel_mss,speed_ms,0,blend_radius_m)
    movel([0.167968, -1.220560, -2.668920, -0.822909, 1.570796, 1.738764],accel_mss,speed_ms,0,blend_radius_m)
    movel([0.168538, -1.217729, -2.670326, -0.824334, 1.570796, 1.739335],accel_mss,speed_ms,0,blend_radius_m)
    movel([0.168667, -1.215028, -2.671659, -0.825703, 1.570796, 1.739464],accel_mss,speed_ms,0,blend_radius_m)
    movel([0.168338, -1.212533, -2.672882, -0.826974, 1.570796, 1.739135],accel_mss,speed_ms,0,blend_radius_m)
    movel([0.167542, -1.210322, -2.673961, -0.828106, 1.570796, 1.738339],accel_mss,speed_ms,0,blend_radius_m)
    movel([0.166271, -1.208476, -2.674857, -0.829056, 1.570796, 1.737068],accel_mss,speed_ms,0,blend_radius_m)
    movel([0.165405, -1.207661, -2.675252, -0.829476, 1.570796, 1.736201],accel_mss,speed_ms,0,blend_radius_m)
    movel([0.164430, -1.206973, -2.675584, -0.829832, 1.570796, 1.735227],accel_mss,speed_ms,0,blend_radius_m)
    movel([0.162198, -1.205984, -2.676061, -0.830344, 1.570796, 1.732994],accel_mss,speed_ms,0,blend_radius_m)
    movel([0.159641, -1.205506, -2.676292, -0.830592, 1.570796, 1.730437],accel_mss,speed_ms,0,blend_radius_m)
    movel([0.156820, -1.205538, -2.676276, -0.830575, 1.570796, 1.727616],accel_mss,speed_ms,0,blend_radius_m)
    movel([0.153804, -1.206068, -2.676021, -0.830300, 1.570796, 1.724600],accel_mss,speed_ms,0,blend_radius_m)
    movel([0.150659, -1.207094, -2.675526, -0.829769, 1.570796, 1.721455],accel_mss,speed_ms,0,blend_radius_m)
    movel([0.147454, -1.208605, -2.674795, -0.828989, 1.570796, 1.718250],accel_mss,speed_ms,0,blend_radius_m)
    movel([0.144260, -1.210585, -2.673833, -0.827971, 1.570796, 1.715057],accel_mss,speed_ms,0,blend_radius_m)
    movel([0.141097, -1.213032, -2.672638, -0.826719, 1.570796, 1.711893],accel_mss,speed_ms,0,blend_radius_m)
    movel([0.138253, -1.215706, -2.671325, -0.825358, 1.570796, 1.709050],accel_mss,speed_ms,0,blend_radius_m)
    movel([0.135764, -1.218555, -2.669917, -0.823918, 1.570796, 1.706560],accel_mss,speed_ms,0,blend_radius_m)
    movel([0.133664, -1.221517, -2.668443, -0.822429, 1.570796, 1.704460],accel_mss,speed_ms,0,blend_radius_m)
    movel([0.131980, -1.224538, -2.666929, -0.820922, 1.570796, 1.702776],accel_mss,speed_ms,0,blend_radius_m)
    movel([0.130744, -1.227570, -2.665400, -0.819419, 1.570796, 1.701540],accel_mss,speed_ms,0,blend_radius_m)
    movel([0.129983, -1.230560, -2.663881, -0.817948, 1.570796, 1.700779],accel_mss,speed_ms,0,blend_radius_m)
    movel([0.129724, -1.233461, -2.662397, -0.816530, 1.570796, 1.700520],accel_mss,speed_ms,0,blend_radius_m)
    movel([0.129934, -1.235684, -2.661254, -0.815451, 1.570796, 1.700730],accel_mss,speed_ms,0,blend_radius_m)
    movel([0.130525, -1.237706, -2.660209, -0.814474, 1.570796, 1.701322],accel_mss,speed_ms,0,blend_radius_m)
    movel([0.131450, -1.239478, -2.659289, -0.813622, 1.570796, 1.702247],accel_mss,speed_ms,0,blend_radius_m)
    movel([0.132666, -1.240957, -2.658519, -0.812913, 1.570796, 1.703462],accel_mss,speed_ms,0,blend_radius_m)
    movel([0.134124, -1.242104, -2.657920, -0.812366, 1.570796, 1.704920],accel_mss,speed_ms,0,blend_radius_m)
    movel([0.135782, -1.242870, -2.657518, -0.812001, 1.570796, 1.706578],accel_mss,speed_ms,0,blend_radius_m)
    movel([0.137600, -1.243214, -2.657338, -0.811837, 1.570796, 1.708396],accel_mss,speed_ms,0,blend_radius_m)
    movel([0.138555, -1.243213, -2.657339, -0.811838, 1.570796, 1.709352],accel_mss,speed_ms,0,blend_radius_m)
    movel([0.139535, -1.243086, -2.657405, -0.811898, 1.570796, 1.710332],accel_mss,speed_ms,0,blend_radius_m)
    movel([0.141303, -1.239677, -2.659186, -0.813526, 1.570796, 1.712099],accel_mss,speed_ms,0,blend_radius_m)
    movel([0.138607, -1.238272, -2.659916, -0.814201, 1.570796, 1.709403],accel_mss,speed_ms,0,blend_radius_m)
    movel([0.136534, -1.236670, -2.660745, -0.814974, 1.570796, 1.707330],accel_mss,speed_ms,0,blend_radius_m)
    movel([0.135733, -1.235790, -2.661199, -0.815399, 1.570796, 1.706529],accel_mss,speed_ms,0,blend_radius_m)
    movel([0.134591, -1.233871, -2.662187, -0.816331, 1.570796, 1.705387],accel_mss,speed_ms,0,blend_radius_m)
    movel([0.134255, -1.232827, -2.662723, -0.816839, 1.570796, 1.705052],accel_mss,speed_ms,0,blend_radius_m)
    movel([0.134077, -1.231723, -2.663287, -0.817378, 1.570796, 1.704874],accel_mss,speed_ms,0,blend_radius_m)
    movel([0.134054, -1.230563, -2.663879, -0.817946, 1.570796, 1.704851],accel_mss,speed_ms,0,blend_radius_m)
    movel([0.134191, -1.229340, -2.664502, -0.818547, 1.570796, 1.704987],accel_mss,speed_ms,0,blend_radius_m)
    movel([0.134481, -1.228057, -2.665153, -0.819179, 1.570796, 1.705277],accel_mss,speed_ms,0,blend_radius_m)
    movel([0.134932, -1.226708, -2.665836, -0.819845, 1.570796, 1.705729],accel_mss,speed_ms,0,blend_radius_m)
    movel([0.135539, -1.225298, -2.666547, -0.820544, 1.570796, 1.706335],accel_mss,speed_ms,0,blend_radius_m)
    movel([0.137231, -1.222276, -2.668063, -0.822049, 1.570796, 1.708028],accel_mss,speed_ms,0,blend_radius_m)
    movel([0.139152, -1.219620, -2.669388, -0.823381, 1.570796, 1.709948],accel_mss,speed_ms,0,blend_radius_m)
    movel([0.141361, -1.217195, -2.670590, -0.824604, 1.570796, 1.712157],accel_mss,speed_ms,0,blend_radius_m)
    movel([0.143791, -1.215046, -2.671650, -0.825693, 1.570796, 1.714588],accel_mss,speed_ms,0,blend_radius_m)
    movel([0.146381, -1.213214, -2.672549, -0.826626, 1.570796, 1.717177],accel_mss,speed_ms,0,blend_radius_m)
    movel([0.149060, -1.211748, -2.673266, -0.827375, 1.570796, 1.719857],accel_mss,speed_ms,0,blend_radius_m)
    movel([0.151762, -1.210691, -2.673782, -0.827917, 1.570796, 1.722558],accel_mss,speed_ms,0,blend_radius_m)
    movel([0.154417, -1.210084, -2.674077, -0.828228, 1.570796, 1.725214],accel_mss,speed_ms,0,blend_radius_m)
    movel([0.156959, -1.209973, -2.674131, -0.828285, 1.570796, 1.727755],accel_mss,speed_ms,0,blend_radius_m)
    movel([0.158199, -1.210118, -2.674060, -0.828211, 1.570796, 1.728995],accel_mss,speed_ms,0,blend_radius_m)
    movel([0.160342, -1.210791, -2.673733, -0.827866, 1.570796, 1.731138],accel_mss,speed_ms,0,blend_radius_m)
    movel([0.161243, -1.211317, -2.673476, -0.827596, 1.570796, 1.732040],accel_mss,speed_ms,0,blend_radius_m)
    movel([0.162708, -1.212733, -2.672785, -0.826872, 1.570796, 1.733504],accel_mss,speed_ms,0,blend_radius_m)
    movel([0.163720, -1.214623, -2.671858, -0.825908, 1.570796, 1.734517],accel_mss,speed_ms,0,blend_radius_m)
    movel([0.164122, -1.216101, -2.671130, -0.825158, 1.570796, 1.734919],accel_mss,speed_ms,0,blend_radius_m)
    movel([0.164273, -1.217652, -2.670364, -0.824373, 1.570796, 1.735070],accel_mss,speed_ms,0,blend_radius_m)
    movel([0.164184, -1.219270, -2.669562, -0.823557, 1.570796, 1.734981],accel_mss,speed_ms,0,blend_radius_m)
    movel([0.163871, -1.220953, -2.668724, -0.822712, 1.570796, 1.734667],accel_mss,speed_ms,0,blend_radius_m)
    movel([0.163341, -1.222691, -2.667856, -0.821842, 1.570796, 1.734138],accel_mss,speed_ms,0,blend_radius_m)
    movel([0.162608, -1.224486, -2.666955, -0.820948, 1.570796, 1.733404],accel_mss,speed_ms,0,blend_radius_m)
    movel([0.161685, -1.226328, -2.666027, -0.820033, 1.570796, 1.732481],accel_mss,speed_ms,0,blend_radius_m)
    movel([0.160585, -1.228213, -2.665074, -0.819102, 1.570796, 1.731381],accel_mss,speed_ms,0,blend_radius_m)
    movel([0.163671, -1.229102, -2.664623, -0.818664, 1.570796, 1.734467],accel_mss,speed_ms,0,blend_radius_m)
    movel([0.165524, -1.226318, -2.666033, -0.820038, 1.570796, 1.736320],accel_mss,speed_ms,0,blend_radius_m)
    speed_ms = 0.005
    # Splitting Linear movement in 4 (instruction 1016: MoveL 952)
    movel([0.165524, -1.223893, -2.664865, -0.823631, 1.570796, 1.736320],accel_mss,speed_ms,0,blend_radius_m)
    movel([0.165524, -1.221483, -2.663693, -0.827213, 1.570796, 1.736320],accel_mss,speed_ms,0,blend_radius_m)
    movel([0.165524, -1.219088, -2.662518, -0.830783, 1.570796, 1.736320],accel_mss,speed_ms,0,blend_radius_m)
    movel([0.165524, -1.216707, -2.661340, -0.834342, 1.570796, 1.736320],accel_mss,speed_ms,0,blend_radius_m)
    speed_ms = 0.040
    # Splitting Linear movement in 8 (instruction 1018: MoveL 953)
    movel([0.167766, -1.217429, -2.660980, -0.833980, 1.570796, 1.738562],accel_mss,speed_ms,0,blend_radius_m)
    movel([0.170001, -1.218157, -2.660617, -0.833616, 1.570796, 1.740797],accel_mss,speed_ms,0,blend_radius_m)
    movel([0.172230, -1.218891, -2.660249, -0.833249, 1.570796, 1.743026],accel_mss,speed_ms,0,blend_radius_m)
    movel([0.174452, -1.219632, -2.659878, -0.832879, 1.570796, 1.745249],accel_mss,speed_ms,0,blend_radius_m)
    movel([0.176668, -1.220379, -2.659503, -0.832507, 1.570796, 1.747465],accel_mss,speed_ms,0,blend_radius_m)
    movel([0.178878, -1.221133, -2.659124, -0.832132, 1.570796, 1.749674],accel_mss,speed_ms,0,blend_radius_m)
    movel([0.181081, -1.221892, -2.658742, -0.831755, 1.570796, 1.751878],accel_mss,speed_ms,0,blend_radius_m)
    movel([0.183278, -1.222659, -2.658355, -0.831375, 1.570796, 1.754074],accel_mss,speed_ms,0,blend_radius_m)
    speed_ms = 0.005
    # Splitting Linear movement in 4 (instruction 1020: MoveL 954)
    movel([0.183278, -1.225033, -2.659527, -0.827829, 1.570796, 1.754074],accel_mss,speed_ms,0,blend_radius_m)
    movel([0.183278, -1.227422, -2.660695, -0.824272, 1.570796, 1.754074],accel_mss,speed_ms,0,blend_radius_m)
    movel([0.183278, -1.229826, -2.661860, -0.820703, 1.570796, 1.754074],accel_mss,speed_ms,0,blend_radius_m)
    movel([0.183278, -1.232244, -2.663021, -0.817124, 1.570796, 1.754074],accel_mss,speed_ms,0,blend_radius_m)
    speed_ms = 0.035
    movel([0.185050, -1.229577, -2.664381, -0.818430, 1.570796, 1.755846],accel_mss,speed_ms,0,blend_radius_m)
    movel([0.186685, -1.226803, -2.665788, -0.819798, 1.570796, 1.757481],accel_mss,speed_ms,0,blend_radius_m)
    movel([0.188167, -1.223940, -2.667230, -0.821219, 1.570796, 1.758964],accel_mss,speed_ms,0,blend_radius_m)
    movel([0.189493, -1.221008, -2.668697, -0.822684, 1.570796, 1.760289],accel_mss,speed_ms,0,blend_radius_m)
    movel([0.190642, -1.218023, -2.670180, -0.824186, 1.570796, 1.761439],accel_mss,speed_ms,0,blend_radius_m)
    movel([0.191604, -1.215008, -2.671669, -0.825713, 1.570796, 1.762401],accel_mss,speed_ms,0,blend_radius_m)
    movel([0.192368, -1.211977, -2.673154, -0.827258, 1.570796, 1.763165],accel_mss,speed_ms,0,blend_radius_m)
    movel([0.192919, -1.208956, -2.674625, -0.828808, 1.570796, 1.763715],accel_mss,speed_ms,0,blend_radius_m)
    movel([0.193243, -1.205961, -2.676072, -0.830355, 1.570796, 1.764039],accel_mss,speed_ms,0,blend_radius_m)
    movel([0.193330, -1.203013, -2.677488, -0.831888, 1.570796, 1.764126],accel_mss,speed_ms,0,blend_radius_m)
    movel([0.193159, -1.200139, -2.678858, -0.833392, 1.570796, 1.763955],accel_mss,speed_ms,0,blend_radius_m)
    movel([0.192720, -1.197359, -2.680176, -0.834855, 1.570796, 1.763517],accel_mss,speed_ms,0,blend_radius_m)
    movel([0.192000, -1.194694, -2.681430, -0.836265, 1.570796, 1.762796],accel_mss,speed_ms,0,blend_radius_m)
    movel([0.190984, -1.192169, -2.682612, -0.837608, 1.570796, 1.761780],accel_mss,speed_ms,0,blend_radius_m)
    movel([0.189658, -1.189810, -2.683710, -0.838870, 1.570796, 1.760454],accel_mss,speed_ms,0,blend_radius_m)
    movel([0.188006, -1.187637, -2.684715, -0.840037, 1.570796, 1.758802],accel_mss,speed_ms,0,blend_radius_m)
    movel([0.186034, -1.185706, -2.685605, -0.841078, 1.570796, 1.756830],accel_mss,speed_ms,0,blend_radius_m)
    movel([0.183805, -1.184084, -2.686349, -0.841956, 1.570796, 1.754602],accel_mss,speed_ms,0,blend_radius_m)
    movel([0.181340, -1.182771, -2.686949, -0.842669, 1.570796, 1.752136],accel_mss,speed_ms,0,blend_radius_m)
    movel([0.178653, -1.181772, -2.687405, -0.843212, 1.570796, 1.749450],accel_mss,speed_ms,0,blend_radius_m)
    movel([0.175765, -1.181086, -2.687717, -0.843586, 1.570796, 1.746561],accel_mss,speed_ms,0,blend_radius_m)
    movel([0.172695, -1.180712, -2.687887, -0.843790, 1.570796, 1.743491],accel_mss,speed_ms,0,blend_radius_m)
    movel([0.169469, -1.180648, -2.687916, -0.843825, 1.570796, 1.740265],accel_mss,speed_ms,0,blend_radius_m)
    movel([0.166102, -1.180893, -2.687805, -0.843692, 1.570796, 1.736898],accel_mss,speed_ms,0,blend_radius_m)
    movel([0.162621, -1.181440, -2.687556, -0.843393, 1.570796, 1.733417],accel_mss,speed_ms,0,blend_radius_m)
    movel([0.159044, -1.182293, -2.687167, -0.842929, 1.570796, 1.729840],accel_mss,speed_ms,0,blend_radius_m)
    movel([0.155393, -1.183442, -2.686643, -0.842304, 1.570796, 1.726189],accel_mss,speed_ms,0,blend_radius_m)
    movel([0.151692, -1.184884, -2.685982, -0.841523, 1.570796, 1.722489],accel_mss,speed_ms,0,blend_radius_m)
    movel([0.147964, -1.186615, -2.685187, -0.840588, 1.570796, 1.718760],accel_mss,speed_ms,0,blend_radius_m)
    movel([0.144226, -1.188625, -2.684258, -0.839505, 1.570796, 1.715023],accel_mss,speed_ms,0,blend_radius_m)
    movel([0.140507, -1.190912, -2.683198, -0.838280, 1.570796, 1.711304],accel_mss,speed_ms,0,blend_radius_m)
    movel([0.136826, -1.193463, -2.682007, -0.836919, 1.570796, 1.707622],accel_mss,speed_ms,0,blend_radius_m)
    movel([0.133191, -1.196280, -2.680684, -0.835425, 1.570796, 1.703987],accel_mss,speed_ms,0,blend_radius_m)
    movel([0.129733, -1.199258, -2.679277, -0.833855, 1.570796, 1.700530],accel_mss,speed_ms,0,blend_radius_m)
    movel([0.126470, -1.202368, -2.677796, -0.832225, 1.570796, 1.697266],accel_mss,speed_ms,0,blend_radius_m)
    movel([0.123412, -1.205590, -2.676251, -0.830548, 1.570796, 1.694208],accel_mss,speed_ms,0,blend_radius_m)
    movel([0.120568, -1.208901, -2.674651, -0.828837, 1.570796, 1.691365],accel_mss,speed_ms,0,blend_radius_m)
    movel([0.117952, -1.212283, -2.673004, -0.827101, 1.570796, 1.688748],accel_mss,speed_ms,0,blend_radius_m)
    movel([0.115566, -1.215719, -2.671318, -0.825351, 1.570796, 1.686363],accel_mss,speed_ms,0,blend_radius_m)
    movel([0.113428, -1.219182, -2.669605, -0.823601, 1.570796, 1.684225],accel_mss,speed_ms,0,blend_radius_m)
    movel([0.111540, -1.222659, -2.667872, -0.821858, 1.570796, 1.682336],accel_mss,speed_ms,0,blend_radius_m)
    movel([0.109910, -1.226133, -2.666126, -0.820130, 1.570796, 1.680707],accel_mss,speed_ms,0,blend_radius_m)
